LIN {X -0.046,Y -453.549,Z 733.557,A 0.000,B 0.000,C 90.000,E1 280.254} C_DIS
LIN {X 0.067,Y -465.639,Z 733.548,A 0.000,B 0.000,C 90.000,E1 278.690} C_DIS
LIN {X -0.179,Y -473.336,Z 733.543,A 0.000,B 0.000,C 90.000,E1 277.701} C_DIS
LIN {X -0.211,Y -478.457,Z 733.538,A 0.000,B 0.000,C 90.000,E1 276.947} C_DIS
LIN {X 0.222,Y -482.858,Z 733.534,A 0.000,B 0.000,C 90.000,E1 276.144} C_DIS
LIN {X -0.212,Y -486.445,Z 733.530,A 0.000,B 0.000,C 90.000,E1 275.448} C_DIS
LIN {X 0.102,Y -487.449,Z 733.529,A 0.000,B 0.000,C 90.000,E1 275.163} C_DIS
LIN {X -0.185,Y -489.129,Z 733.526,A 0.000,B 0.000,C 90.000,E1 274.702} C_DIS
LIN {X -0.017,Y -490.429,Z 733.523,A 0.000,B 0.000,C 90.000,E1 274.188} C_DIS
LIN {X 0.198,Y -491.326,Z 733.521,A 0.000,B 0.000,C 90.000,E1 273.669} C_DIS
LIN {X -0.101,Y -491.778,Z 733.518,A 0.000,B 0.000,C 90.000,E1 273.212} C_DIS
LIN {X 0.124,Y -491.880,Z 733.515,A 0.000,B 0.000,C 90.000,E1 272.694} C_DIS
LIN {X -0.164,Y -491.605,Z 733.512,A 0.000,B 0.000,C 90.000,E1 272.236} C_DIS
LIN {X 0.057,Y -490.893,Z 733.510,A 0.000,B 0.000,C 90.000,E1 271.718} C_DIS
LIN {X -0.231,Y -489.791,Z 733.507,A 0.000,B 0.000,C 90.000,E1 271.260} C_DIS
LIN {X -0.031,Y -488.272,Z 733.504,A 0.000,B 0.000,C 90.000,E1 270.745} C_DIS
LIN {X 0.162,Y -486.222,Z 733.501,A 0.000,B 0.000,C 90.000,E1 270.229} C_DIS
LIN {X -0.139,Y -483.595,Z 733.499,A 0.000,B 0.000,C 90.000,E1 269.771} C_DIS
LIN {X 0.026,Y -480.228,Z 733.496,A 0.000,B 0.000,C 90.000,E1 269.255} C_DIS
LIN {X 0.171,Y -476.025,Z 733.493,A 0.000,B 0.000,C 90.000,E1 268.740} C_DIS
LIN {X -0.006,Y -473.521,Z 733.492,A 0.000,B 0.000,C 90.000,E1 268.511} C_DIS
LIN {X -0.139,Y -467.895,Z 733.489,A 0.000,B 0.000,C 90.000,E1 268.051} C_DIS
LIN {X 0.151,Y -461.751,Z 733.487,A 0.000,B 0.000,C 90.000,E1 267.593} C_DIS
LIN {X 0.008,Y -455.030,Z 733.485,A 0.000,B 0.000,C 90.000,E1 267.249} C_DIS
LIN {X -0.087,Y -447.759,Z 733.483,A 0.000,B 0.000,C 90.000,E1 266.963} C_DIS
LIN {X -0.124,Y -439.978,Z 733.482,A 0.000,B 0.000,C 90.000,E1 266.731} C_DIS
LIN {X -0.126,Y -431.439,Z 733.481,A 0.000,B 0.000,C 90.000,E1 266.560} C_DIS
LIN {X 0.048,Y -423.516,Z 733.480,A 0.000,B 0.000,C 90.000,E1 266.445} C_DIS
LIN {X -0.116,Y -418.864,Z 733.480,A 0.000,B 0.000,C 90.000,E1 266.445} C_DIS
LIN {X -0.086,Y -180.942,Z 733.480,A 0.000,B 0.000,C 90.000,E1 266.445} C_DIS
LIN {X -0.075,Y -180.767,Z 733.471,A 0.000,B 0.000,C 90.000,E1 264.723} C_DIS
LIN {X -0.004,Y -178.861,Z 733.442,A 0.000,B 0.000,C 90.000,E1 259.634} C_DIS
LIN {X 0.067,Y -175.904,Z 733.414,A 0.000,B 0.000,C 90.000,E1 254.519} C_DIS
LIN {X 0.006,Y -174.587,Z 733.405,A 0.000,B 0.000,C 90.000,E1 252.834} C_DIS
LIN {X 0.041,Y -171.570,Z 733.381,A 0.000,B 0.000,C 90.000,E1 248.539} C_DIS
LIN {X 0.023,Y -167.793,Z 733.357,A 0.000,B 0.000,C 90.000,E1 244.229} C_DIS
LIN {X 0.037,Y -166.509,Z 733.347,A 0.000,B 0.000,C 90.000,E1 242.487} C_DIS
LIN {X 0.032,Y -163.218,Z 733.328,A 0.000,B 0.000,C 90.000,E1 238.997} C_DIS
LIN {X -0.003,Y -161.183,Z 733.313,A 0.000,B 0.000,C 90.000,E1 236.373} C_DIS
LIN {X -0.003,Y -157.196,Z 733.289,A 0.000,B 0.000,C 90.000,E1 231.949} C_DIS
LIN {X 0.043,Y -155.924,Z 733.279,A 0.000,B 0.000,C 90.000,E1 230.150} C_DIS
LIN {X -0.007,Y -152.175,Z 733.254,A 0.000,B 0.000,C 90.000,E1 225.688} C_DIS
LIN {X 0.008,Y -150.423,Z 733.239,A 0.000,B 0.000,C 90.000,E1 222.975} C_DIS
LIN {X -0.066,Y -147.151,Z 733.214,A 0.000,B 0.000,C 90.000,E1 218.463} C_DIS
LIN {X 0.021,Y -145.165,Z 733.193,A 0.000,B 0.000,C 90.000,E1 214.771} C_DIS
LIN {X -0.063,Y -142.318,Z 733.163,A 0.000,B 0.000,C 90.000,E1 209.283} C_DIS
LIN {X 0.058,Y -141.708,Z 733.152,A 0.000,B 0.000,C 90.000,E1 207.385} C_DIS
LIN {X -0.020,Y -139.470,Z 733.116,A 0.000,B 0.000,C 90.000,E1 200.918} C_DIS
LIN {X 0.034,Y -139.202,Z 733.106,A 0.000,B 0.000,C 90.000,E1 199.033} C_DIS
LIN {X -0.039,Y -138.329,Z 733.054,A 0.000,B 0.000,C 90.000,E1 189.726} C_DIS
LIN {X -0.036,Y -139.441,Z 733.007,A 0.000,B 0.000,C 90.000,E1 181.318} C_DIS
LIN {X 0.043,Y -140.976,Z 732.976,A 0.000,B 0.000,C 90.000,E1 175.698} C_DIS
LIN {X -0.007,Y -142.731,Z 732.956,A 0.000,B 0.000,C 90.000,E1 172.008} C_DIS
LIN {X -0.050,Y -145.119,Z 732.930,A 0.000,B 0.000,C 90.000,E1 167.409} C_DIS
LIN {X -0.055,Y -147.743,Z 732.910,A 0.000,B 0.000,C 90.000,E1 163.740} C_DIS
LIN {X 0.026,Y -150.409,Z 732.889,A 0.000,B 0.000,C 90.000,E1 160.061} C_DIS
LIN {X 0.042,Y -153.847,Z 732.869,A 0.000,B 0.000,C 90.000,E1 156.433} C_DIS
LIN {X -0.041,Y -157.258,Z 732.849,A 0.000,B 0.000,C 90.000,E1 152.871} C_DIS
LIN {X 0.037,Y -161.432,Z 732.829,A 0.000,B 0.000,C 90.000,E1 149.282} C_DIS
LIN {X 0.044,Y -165.633,Z 732.810,A 0.000,B 0.000,C 90.000,E1 145.754} C_DIS
LIN {X 0.027,Y -170.564,Z 732.790,A 0.000,B 0.000,C 90.000,E1 142.271} C_DIS
LIN {X -0.065,Y -175.443,Z 732.771,A 0.000,B 0.000,C 90.000,E1 138.852} C_DIS
LIN {X 0.051,Y -181.066,Z 732.752,A 0.000,B 0.000,C 90.000,E1 135.405} C_DIS
LIN {X -0.084,Y -186.504,Z 732.734,A 0.000,B 0.000,C 90.000,E1 132.081} C_DIS
LIN {X 0.015,Y -191.572,Z 732.718,A 0.000,B 0.000,C 90.000,E1 129.277} C_DIS
LIN {X -0.056,Y -191.740,Z 732.718,A 0.000,B 0.000,C 90.000,E1 129.197} C_DIS
LIN {X -0.129,Y -290.705,Z 732.718,A 0.000,B 0.000,C 90.000,E1 129.197} C_DIS
LIN {X 0.010,Y -291.831,Z 732.718,A 0.000,B 0.000,C 90.000,E1 129.152} C_DIS
LIN {X -0.060,Y -296.587,Z 732.716,A 0.000,B 0.000,C 90.000,E1 128.955} C_DIS
LIN {X -0.089,Y -299.097,Z 732.715,A 0.000,B 0.000,C 90.000,E1 128.749} C_DIS
LIN {X -0.093,Y -302.912,Z 732.712,A 0.000,B 0.000,C 90.000,E1 128.257} C_DIS
LIN {X 0.096,Y -304.694,Z 732.711,A 0.000,B 0.000,C 90.000,E1 127.890} C_DIS
LIN {X 0.042,Y -306.088,Z 732.709,A 0.000,B 0.000,C 90.000,E1 127.569} C_DIS
LIN {X -0.168,Y -309.945,Z 732.701,A 0.000,B 0.000,C 90.000,E1 126.297} C_DIS
LIN {X -0.051,Y -320.114,Z 732.683,A 0.000,B 0.000,C 90.000,E1 123.038} C_DIS
LIN {X -0.047,Y -330.586,Z 732.668,A 0.000,B 0.000,C 90.000,E1 120.178} C_DIS
LIN {X -0.131,Y -342.421,Z 732.652,A 0.000,B 0.000,C 90.000,E1 117.385} C_DIS
LIN {X -0.181,Y -355.717,Z 732.637,A 0.000,B 0.000,C 90.000,E1 114.643} C_DIS
LIN {X 0.103,Y -368.862,Z 732.623,A 0.000,B 0.000,C 90.000,E1 112.206} C_DIS
LIN {X -0.031,Y -383.352,Z 732.610,A 0.000,B 0.000,C 90.000,E1 109.885} C_DIS
LIN {X 0.074,Y -399.291,Z 732.598,A 0.000,B 0.000,C 90.000,E1 107.583} C_DIS
LIN {X -0.051,Y -416.796,Z 732.585,A 0.000,B 0.000,C 90.000,E1 105.371} C_DIS
LIN {X 0.159,Y -435.964,Z 732.573,A 0.000,B 0.000,C 90.000,E1 103.175} C_DIS
LIN {X -0.137,Y -456.118,Z 732.562,A 0.000,B 0.000,C 90.000,E1 101.186} C_DIS
LIN {X 0.211,Y -468.863,Z 732.555,A 0.000,B 0.000,C 90.000,E1 99.962} C_DIS
LIN {X 0.182,Y -470.793,Z 732.554,A 0.000,B 0.000,C 90.000,E1 99.726} C_DIS
LIN {X 0.073,Y -472.261,Z 732.553,A 0.000,B 0.000,C 90.000,E1 99.500} C_DIS
LIN {X 0.252,Y -474.285,Z 732.550,A 0.000,B 0.000,C 90.000,E1 98.973} C_DIS
LIN {X -0.104,Y -475.176,Z 732.547,A 0.000,B 0.000,C 90.000,E1 98.511} C_DIS
LIN {X 0.022,Y -475.088,Z 732.544,A 0.000,B 0.000,C 90.000,E1 97.992} C_DIS
LIN {X 0.156,Y -474.014,Z 732.542,A 0.000,B 0.000,C 90.000,E1 97.473} C_DIS
LIN {X 0.018,Y -473.060,Z 732.540,A 0.000,B 0.000,C 90.000,E1 97.239} C_DIS
LIN {X -0.122,Y -471.768,Z 732.539,A 0.000,B 0.000,C 90.000,E1 97.004} C_DIS
LIN {X 0.005,Y -453.891,Z 732.523,A 0.000,B 0.000,C 90.000,E1 94.188} C_DIS
LIN {X -0.165,Y -439.054,Z 732.509,A 0.000,B 0.000,C 90.000,E1 91.604} C_DIS
LIN {X -0.208,Y -431.544,Z 732.501,A 0.000,B 0.000,C 90.000,E1 90.286} C_DIS
LIN {X 0.015,Y -419.099,Z 732.490,A 0.000,B 0.000,C 90.000,E1 88.108} C_DIS
LIN {X -0.140,Y -408.057,Z 732.479,A 0.000,B 0.000,C 90.000,E1 86.216} C_DIS
LIN {X -0.063,Y -396.902,Z 732.468,A 0.000,B 0.000,C 90.000,E1 84.261} C_DIS
LIN {X -0.132,Y -384.313,Z 732.456,A 0.000,B 0.000,C 90.000,E1 82.008} C_DIS
LIN {X -0.068,Y -372.095,Z 732.443,A 0.000,B 0.000,C 90.000,E1 79.690} C_DIS
LIN {X -0.123,Y -358.888,Z 732.428,A 0.000,B 0.000,C 90.000,E1 77.048} C_DIS
LIN {X -0.046,Y -348.945,Z 732.416,A 0.000,B 0.000,C 90.000,E1 74.936} C_DIS
LIN {X -0.032,Y -336.383,Z 732.401,A 0.000,B 0.000,C 90.000,E1 72.181} C_DIS
LIN {X -0.140,Y -324.350,Z 732.385,A 0.000,B 0.000,C 90.000,E1 69.390} C_DIS
LIN {X -0.011,Y -312.017,Z 732.368,A 0.000,B 0.000,C 90.000,E1 66.177} C_DIS
LIN {X -0.012,Y -301.168,Z 732.350,A 0.000,B 0.000,C 90.000,E1 62.922} C_DIS
LIN {X -0.049,Y -291.225,Z 732.331,A 0.000,B 0.000,C 90.000,E1 59.616} C_DIS
LIN {X -0.008,Y -283.697,Z 732.316,A 0.000,B 0.000,C 90.000,E1 56.914} C_DIS
LIN {X -0.076,Y -276.550,Z 732.301,A 0.000,B 0.000,C 90.000,E1 54.196} C_DIS
LIN {X -0.001,Y -269.411,Z 732.286,A 0.000,B 0.000,C 90.000,E1 51.412} C_DIS
LIN {X 0.051,Y -263.888,Z 732.274,A 0.000,B 0.000,C 90.000,E1 49.299} C_DIS
LIN {X 0.067,Y -256.395,Z 732.258,A 0.000,B 0.000,C 90.000,E1 46.458} C_DIS
LIN {X -0.145,Y -250.679,Z 732.246,A 0.000,B 0.000,C 90.000,E1 44.352} C_DIS
LIN {X 0.068,Y -244.854,Z 732.234,A 0.000,B 0.000,C 90.000,E1 42.123} C_DIS
LIN {X 0.019,Y -238.963,Z 732.222,A 0.000,B 0.000,C 90.000,E1 39.930} C_DIS
LIN {X -0.061,Y -229.499,Z 732.201,A 0.000,B 0.000,C 90.000,E1 36.217} C_DIS
LIN {X -0.085,Y -220.772,Z 732.180,A 0.000,B 0.000,C 90.000,E1 32.418} C_DIS
LIN {X 0.074,Y -214.464,Z 732.163,A 0.000,B 0.000,C 90.000,E1 29.283} C_DIS
LIN {X 0.044,Y -208.878,Z 732.145,A 0.000,B 0.000,C 90.000,E1 26.155} C_DIS
LIN {X -0.032,Y -202.897,Z 732.123,A 0.000,B 0.000,C 90.000,E1 22.206} C_DIS
LIN {X -0.018,Y -198.172,Z 732.101,A 0.000,B 0.000,C 90.000,E1 18.181} C_DIS
LIN {X -0.014,Y -194.509,Z 732.078,A 0.000,B 0.000,C 90.000,E1 14.120} C_DIS
LIN {X -0.020,Y -191.545,Z 732.051,A 0.000,B 0.000,C 90.000,E1 9.208} C_DIS
LIN {X -0.029,Y -191.025,Z 731.974,A 0.000,B 0.000,C 90.000,E1 355.412} C_DIS
LIN {X 0.080,Y -193.620,Z 731.947,A 0.000,B 0.000,C 90.000,E1 350.443} C_DIS
LIN {X 0.087,Y -196.990,Z 731.924,A 0.000,B 0.000,C 90.000,E1 346.353} C_DIS
LIN {X 0.047,Y -201.312,Z 731.902,A 0.000,B 0.000,C 90.000,E1 342.308} C_DIS
LIN {X 0.073,Y -206.533,Z 731.879,A 0.000,B 0.000,C 90.000,E1 338.284} C_DIS
LIN {X 0.008,Y -212.775,Z 731.857,A 0.000,B 0.000,C 90.000,E1 334.332} C_DIS
LIN {X 0.027,Y -219.597,Z 731.836,A 0.000,B 0.000,C 90.000,E1 330.411} C_DIS
LIN {X 0.046,Y -227.020,Z 731.814,A 0.000,B 0.000,C 90.000,E1 326.548} C_DIS
LIN {X -0.007,Y -235.102,Z 731.793,A 0.000,B 0.000,C 90.000,E1 322.763} C_DIS
LIN {X 0.058,Y -243.917,Z 731.772,A 0.000,B 0.000,C 90.000,E1 319.013} C_DIS
LIN {X -0.021,Y -253.550,Z 731.752,A 0.000,B 0.000,C 90.000,E1 315.364} C_DIS
LIN {X 0.055,Y -264.373,Z 731.732,A 0.000,B 0.000,C 90.000,E1 311.757} C_DIS
LIN {X -0.002,Y -276.186,Z 731.713,A 0.000,B 0.000,C 90.000,E1 308.257} C_DIS
LIN {X 0.030,Y -289.374,Z 731.693,A 0.000,B 0.000,C 90.000,E1 304.818} C_DIS
LIN {X 0.067,Y -304.184,Z 731.675,A 0.000,B 0.000,C 90.000,E1 301.465} C_DIS
LIN {X -0.087,Y -315.631,Z 731.662,A 0.000,B 0.000,C 90.000,E1 299.205} C_DIS
LIN {X 0.145,Y -333.522,Z 731.644,A 0.000,B 0.000,C 90.000,E1 295.976} C_DIS
LIN {X 0.052,Y -350.964,Z 731.629,A 0.000,B 0.000,C 90.000,E1 293.206} C_DIS
LIN {X -0.120,Y -373.760,Z 731.611,A 0.000,B 0.000,C 90.000,E1 289.939} C_DIS
LIN {X 0.126,Y -392.212,Z 731.598,A 0.000,B 0.000,C 90.000,E1 287.583} C_DIS
LIN {X 0.054,Y -406.448,Z 731.588,A 0.000,B 0.000,C 90.000,E1 285.898} C_DIS
LIN {X 0.012,Y -420.554,Z 731.579,A 0.000,B 0.000,C 90.000,E1 284.245} C_DIS
LIN {X 0.082,Y -432.003,Z 731.572,A 0.000,B 0.000,C 90.000,E1 282.883} C_DIS
LIN {X 0.200,Y -442.999,Z 731.564,A 0.000,B 0.000,C 90.000,E1 281.535} C_DIS
LIN {X -0.051,Y -453.387,Z 731.557,A 0.000,B 0.000,C 90.000,E1 280.254} C_DIS
LIN {X 0.130,Y -465.479,Z 731.548,A 0.000,B 0.000,C 90.000,E1 278.681} C_DIS
LIN {X -0.190,Y -473.188,Z 731.543,A 0.000,B 0.000,C 90.000,E1 277.701} C_DIS
LIN {X 0.253,Y -478.317,Z 731.538,A 0.000,B 0.000,C 90.000,E1 276.891} C_DIS
LIN {X 0.209,Y -482.707,Z 731.534,A 0.000,B 0.000,C 90.000,E1 276.144} C_DIS
LIN {X 0.258,Y -486.253,Z 731.530,A 0.000,B 0.000,C 90.000,E1 275.391} C_DIS
LIN {X 0.087,Y -487.248,Z 731.529,A 0.000,B 0.000,C 90.000,E1 275.163} C_DIS
LIN {X -0.200,Y -488.920,Z 731.526,A 0.000,B 0.000,C 90.000,E1 274.702} C_DIS
LIN {X -0.035,Y -490.200,Z 731.523,A 0.000,B 0.000,C 90.000,E1 274.188} C_DIS
LIN {X 0.180,Y -491.070,Z 731.521,A 0.000,B 0.000,C 90.000,E1 273.669} C_DIS
LIN {X -0.120,Y -491.497,Z 731.518,A 0.000,B 0.000,C 90.000,E1 273.212} C_DIS
LIN {X 0.103,Y -491.580,Z 731.515,A 0.000,B 0.000,C 90.000,E1 272.694} C_DIS
LIN {X -0.187,Y -491.309,Z 731.512,A 0.000,B 0.000,C 90.000,E1 272.236} C_DIS
LIN {X 0.033,Y -490.597,Z 731.510,A 0.000,B 0.000,C 90.000,E1 271.718} C_DIS
LIN {X 0.233,Y -489.509,Z 731.507,A 0.000,B 0.000,C 90.000,E1 271.203} C_DIS
LIN {X -0.059,Y -488.013,Z 731.504,A 0.000,B 0.000,C 90.000,E1 270.745} C_DIS
LIN {X 0.133,Y -486.001,Z 731.501,A 0.000,B 0.000,C 90.000,E1 270.229} C_DIS
LIN {X -0.168,Y -483.404,Z 731.499,A 0.000,B 0.000,C 90.000,E1 269.771} C_DIS
LIN {X -0.004,Y -480.098,Z 731.496,A 0.000,B 0.000,C 90.000,E1 269.255} C_DIS
LIN {X 0.139,Y -475.872,Z 731.493,A 0.000,B 0.000,C 90.000,E1 268.740} C_DIS
LIN {X -0.213,Y -470.568,Z 731.490,A 0.000,B 0.000,C 90.000,E1 268.282} C_DIS
LIN {X -0.220,Y -467.738,Z 731.489,A 0.000,B 0.000,C 90.000,E1 268.051} C_DIS
LIN {X 0.044,Y -461.530,Z 731.487,A 0.000,B 0.000,C 90.000,E1 267.593} C_DIS
LIN {X -0.109,Y -454.863,Z 731.485,A 0.000,B 0.000,C 90.000,E1 267.249} C_DIS
LIN {X -0.084,Y -451.037,Z 731.484,A 0.000,B 0.000,C 90.000,E1 267.078} C_DIS
LIN {X 0.095,Y -443.345,Z 731.482,A 0.000,B 0.000,C 90.000,E1 266.788} C_DIS
LIN {X -0.147,Y -434.887,Z 731.481,A 0.000,B 0.000,C 90.000,E1 266.617} C_DIS
LIN {X 0.128,Y -425.733,Z 731.480,A 0.000,B 0.000,C 90.000,E1 266.445} C_DIS
LIN {X -0.198,Y -419.011,Z 731.480,A 0.000,B 0.000,C 90.000,E1 266.445} C_DIS
LIN {X 0.060,Y -180.942,Z 731.480,A 0.000,B 0.000,C 90.000,E1 266.388} C_DIS
LIN {X 0.071,Y -180.762,Z 731.470,A 0.000,B 0.000,C 90.000,E1 264.666} C_DIS
LIN {X -0.038,Y -178.856,Z 731.442,A 0.000,B 0.000,C 90.000,E1 259.634} C_DIS
LIN {X 0.034,Y -175.900,Z 731.414,A 0.000,B 0.000,C 90.000,E1 254.519} C_DIS
LIN {X -0.027,Y -174.578,Z 731.405,A 0.000,B 0.000,C 90.000,E1 252.834} C_DIS
LIN {X 0.007,Y -171.561,Z 731.381,A 0.000,B 0.000,C 90.000,E1 248.539} C_DIS
LIN {X -0.010,Y -167.785,Z 731.357,A 0.000,B 0.000,C 90.000,E1 244.229} C_DIS
LIN {X 0.005,Y -166.499,Z 731.347,A 0.000,B 0.000,C 90.000,E1 242.487} C_DIS
LIN {X 0.000,Y -163.208,Z 731.328,A 0.000,B 0.000,C 90.000,E1 238.997} C_DIS
LIN {X -0.035,Y -161.172,Z 731.313,A 0.000,B 0.000,C 90.000,E1 236.373} C_DIS
LIN {X 0.089,Y -157.186,Z 731.289,A 0.000,B 0.000,C 90.000,E1 231.904} C_DIS
LIN {X 0.012,Y -155.916,Z 731.279,A 0.000,B 0.000,C 90.000,E1 230.150} C_DIS
LIN {X 0.069,Y -152.167,Z 731.254,A 0.000,B 0.000,C 90.000,E1 225.648} C_DIS
LIN {X -0.023,Y -150.415,Z 731.239,A 0.000,B 0.000,C 90.000,E1 222.975} C_DIS
LIN {X 0.019,Y -147.144,Z 731.214,A 0.000,B 0.000,C 90.000,E1 218.418} C_DIS
LIN {X 0.016,Y -145.703,Z 731.198,A 0.000,B 0.000,C 90.000,E1 215.678} C_DIS
LIN {X 0.023,Y -143.085,Z 731.173,A 0.000,B 0.000,C 90.000,E1 211.082} C_DIS
LIN {X 0.029,Y -141.703,Z 731.152,A 0.000,B 0.000,C 90.000,E1 207.385} C_DIS
LIN {X -0.049,Y -139.468,Z 731.116,A 0.000,B 0.000,C 90.000,E1 200.918} C_DIS
LIN {X 0.005,Y -139.201,Z 731.106,A 0.000,B 0.000,C 90.000,E1 199.033} C_DIS
LIN {X 0.068,Y -138.328,Z 731.054,A 0.000,B 0.000,C 90.000,E1 189.670} C_DIS
LIN {X -0.066,Y -139.443,Z 731.007,A 0.000,B 0.000,C 90.000,E1 181.318} C_DIS
LIN {X 0.014,Y -140.981,Z 730.976,A 0.000,B 0.000,C 90.000,E1 175.698} C_DIS
LIN {X -0.036,Y -142.736,Z 730.956,A 0.000,B 0.000,C 90.000,E1 172.008} C_DIS
LIN {X 0.062,Y -145.127,Z 730.930,A 0.000,B 0.000,C 90.000,E1 167.353} C_DIS
LIN {X 0.056,Y -147.750,Z 730.909,A 0.000,B 0.000,C 90.000,E1 163.685} C_DIS
LIN {X -0.004,Y -150.419,Z 730.889,A 0.000,B 0.000,C 90.000,E1 160.061} C_DIS
LIN {X 0.010,Y -153.859,Z 730.869,A 0.000,B 0.000,C 90.000,E1 156.433} C_DIS
LIN {X -0.072,Y -157.270,Z 730.849,A 0.000,B 0.000,C 90.000,E1 152.871} C_DIS
LIN {X 0.005,Y -161.447,Z 730.829,A 0.000,B 0.000,C 90.000,E1 149.282} C_DIS
LIN {X 0.012,Y -165.648,Z 730.810,A 0.000,B 0.000,C 90.000,E1 145.754} C_DIS
LIN {X -0.006,Y -170.581,Z 730.790,A 0.000,B 0.000,C 90.000,E1 142.271} C_DIS
LIN {X -0.099,Y -175.459,Z 730.771,A 0.000,B 0.000,C 90.000,E1 138.852} C_DIS
LIN {X 0.016,Y -181.082,Z 730.752,A 0.000,B 0.000,C 90.000,E1 135.405} C_DIS
LIN {X 0.007,Y -186.523,Z 730.734,A 0.000,B 0.000,C 90.000,E1 132.043} C_DIS
LIN {X -0.020,Y -191.589,Z 730.718,A 0.000,B 0.000,C 90.000,E1 129.277} C_DIS
LIN {X 0.007,Y -191.708,Z 730.718,A 0.000,B 0.000,C 90.000,E1 129.197} C_DIS
LIN {X -0.024,Y -290.454,Z 730.718,A 0.000,B 0.000,C 90.000,E1 129.197} C_DIS
LIN {X 0.143,Y -292.896,Z 730.717,A 0.000,B 0.000,C 90.000,E1 129.116} C_DIS
LIN {X 0.116,Y -296.939,Z 730.716,A 0.000,B 0.000,C 90.000,E1 128.910} C_DIS
LIN {X -0.144,Y -299.327,Z 730.715,A 0.000,B 0.000,C 90.000,E1 128.749} C_DIS
LIN {X -0.075,Y -303.151,Z 730.712,A 0.000,B 0.000,C 90.000,E1 128.222} C_DIS
LIN {X -0.073,Y -304.863,Z 730.710,A 0.000,B 0.000,C 90.000,E1 127.890} C_DIS
LIN {X 0.116,Y -306.203,Z 730.709,A 0.000,B 0.000,C 90.000,E1 127.523} C_DIS
LIN {X -0.018,Y -314.920,Z 730.692,A 0.000,B 0.000,C 90.000,E1 124.612} C_DIS
LIN {X 0.102,Y -325.861,Z 730.674,A 0.000,B 0.000,C 90.000,E1 121.386} C_DIS
LIN {X 0.052,Y -337.094,Z 730.659,A 0.000,B 0.000,C 90.000,E1 118.565} C_DIS
LIN {X 0.018,Y -349.741,Z 730.643,A 0.000,B 0.000,C 90.000,E1 115.796} C_DIS
LIN {X -0.027,Y -362.264,Z 730.630,A 0.000,B 0.000,C 90.000,E1 113.387} C_DIS
LIN {X -0.196,Y -376.086,Z 730.617,A 0.000,B 0.000,C 90.000,E1 111.046} C_DIS
LIN {X -0.155,Y -391.304,Z 730.604,A 0.000,B 0.000,C 90.000,E1 108.725} C_DIS
LIN {X 0.019,Y -408.030,Z 730.591,A 0.000,B 0.000,C 90.000,E1 106.441} C_DIS
LIN {X -0.006,Y -426.384,Z 730.579,A 0.000,B 0.000,C 90.000,E1 104.245} C_DIS
LIN {X 0.128,Y -446.191,Z 730.567,A 0.000,B 0.000,C 90.000,E1 102.119} C_DIS
LIN {X 0.022,Y -469.054,Z 730.555,A 0.000,B 0.000,C 90.000,E1 99.962} C_DIS
LIN {X -0.025,Y -470.957,Z 730.554,A 0.000,B 0.000,C 90.000,E1 99.726} C_DIS
LIN {X -0.152,Y -472.403,Z 730.553,A 0.000,B 0.000,C 90.000,E1 99.500} C_DIS
LIN {X 0.027,Y -474.369,Z 730.550,A 0.000,B 0.000,C 90.000,E1 98.973} C_DIS
LIN {X 0.141,Y -475.214,Z 730.547,A 0.000,B 0.000,C 90.000,E1 98.454} C_DIS
LIN {X -0.203,Y -475.082,Z 730.544,A 0.000,B 0.000,C 90.000,E1 97.992} C_DIS
LIN {X -0.006,Y -473.962,Z 730.541,A 0.000,B 0.000,C 90.000,E1 97.466} C_DIS
LIN {X -0.206,Y -472.980,Z 730.540,A 0.000,B 0.000,C 90.000,E1 97.239} C_DIS
LIN {X 0.122,Y -471.654,Z 730.539,A 0.000,B 0.000,C 90.000,E1 96.947} C_DIS
LIN {X 0.040,Y -452.227,Z 730.522,A 0.000,B 0.000,C 90.000,E1 93.898} C_DIS
LIN {X 0.059,Y -438.929,Z 730.509,A 0.000,B 0.000,C 90.000,E1 91.547} C_DIS
LIN {X 0.010,Y -431.419,Z 730.501,A 0.000,B 0.000,C 90.000,E1 90.229} C_DIS
LIN {X 0.095,Y -420.536,Z 730.491,A 0.000,B 0.000,C 90.000,E1 88.339} C_DIS
LIN {X -0.097,Y -411.123,Z 730.482,A 0.000,B 0.000,C 90.000,E1 86.731} C_DIS
LIN {X 0.015,Y -400.009,Z 730.471,A 0.000,B 0.000,C 90.000,E1 84.780} C_DIS
LIN {X -0.038,Y -388.917,Z 730.460,A 0.000,B 0.000,C 90.000,E1 82.818} C_DIS
LIN {X 0.089,Y -375.106,Z 730.446,A 0.000,B 0.000,C 90.000,E1 80.218} C_DIS
LIN {X -0.004,Y -360.315,Z 730.429,A 0.000,B 0.000,C 90.000,E1 77.297} C_DIS
LIN {X 0.199,Y -348.938,Z 730.416,A 0.000,B 0.000,C 90.000,E1 74.866} C_DIS
LIN {X 0.112,Y -336.392,Z 730.401,A 0.000,B 0.000,C 90.000,E1 72.127} C_DIS
LIN {X -0.006,Y -324.388,Z 730.385,A 0.000,B 0.000,C 90.000,E1 69.337} C_DIS
LIN {X -0.098,Y -313.255,Z 730.369,A 0.000,B 0.000,C 90.000,E1 66.485} C_DIS
LIN {X -0.090,Y -303.370,Z 730.353,A 0.000,B 0.000,C 90.000,E1 63.563} C_DIS
LIN {X -0.050,Y -293.340,Z 730.335,A 0.000,B 0.000,C 90.000,E1 60.255} C_DIS
LIN {X -0.099,Y -285.776,Z 730.320,A 0.000,B 0.000,C 90.000,E1 57.582} C_DIS
LIN {X 0.022,Y -276.791,Z 730.301,A 0.000,B 0.000,C 90.000,E1 54.149} C_DIS
LIN {X 0.082,Y -271.470,Z 730.289,A 0.000,B 0.000,C 90.000,E1 52.065} C_DIS
LIN {X 0.000,Y -266.029,Z 730.278,A 0.000,B 0.000,C 90.000,E1 49.989} C_DIS
LIN {X -0.011,Y -260.411,Z 730.266,A 0.000,B 0.000,C 90.000,E1 47.877} C_DIS
LIN {X 0.030,Y -254.806,Z 730.254,A 0.000,B 0.000,C 90.000,E1 45.729} C_DIS
LIN {X -0.028,Y -249.029,Z 730.242,A 0.000,B 0.000,C 90.000,E1 43.581} C_DIS
LIN {X -0.012,Y -243.173,Z 730.230,A 0.000,B 0.000,C 90.000,E1 41.391} C_DIS
LIN {X -0.124,Y -235.311,Z 730.214,A 0.000,B 0.000,C 90.000,E1 38.463} C_DIS
LIN {X -0.076,Y -226.129,Z 730.193,A 0.000,B 0.000,C 90.000,E1 34.692} C_DIS
LIN {X 0.077,Y -219.325,Z 730.176,A 0.000,B 0.000,C 90.000,E1 31.592} C_DIS
LIN {X 0.083,Y -213.153,Z 730.158,A 0.000,B 0.000,C 90.000,E1 28.487} C_DIS
LIN {X 0.109,Y -207.762,Z 730.141,A 0.000,B 0.000,C 90.000,E1 25.335} C_DIS
LIN {X -0.071,Y -203.043,Z 730.123,A 0.000,B 0.000,C 90.000,E1 22.206} C_DIS
LIN {X -0.053,Y -198.302,Z 730.101,A 0.000,B 0.000,C 90.000,E1 18.181} C_DIS
LIN {X -0.044,Y -194.624,Z 730.078,A 0.000,B 0.000,C 90.000,E1 14.120} C_DIS
LIN {X -0.046,Y -191.640,Z 730.051,A 0.000,B 0.000,C 90.000,E1 9.208} C_DIS
LIN {X 0.044,Y -190.829,Z 729.979,A 0.000,B 0.000,C 90.000,E1 356.216} C_DIS
LIN {X 0.088,Y -193.734,Z 729.947,A 0.000,B 0.000,C 90.000,E1 350.443} C_DIS
LIN {X -0.094,Y -197.092,Z 729.924,A 0.000,B 0.000,C 90.000,E1 346.408} C_DIS
LIN {X 0.061,Y -201.422,Z 729.902,A 0.000,B 0.000,C 90.000,E1 342.308} C_DIS
LIN {X 0.092,Y -206.646,Z 729.880,A 0.000,B 0.000,C 90.000,E1 338.284} C_DIS
LIN {X 0.030,Y -212.868,Z 729.857,A 0.000,B 0.000,C 90.000,E1 334.332} C_DIS
LIN {X 0.053,Y -219.668,Z 729.836,A 0.000,B 0.000,C 90.000,E1 330.411} C_DIS
LIN {X -0.050,Y -227.083,Z 729.814,A 0.000,B 0.000,C 90.000,E1 326.580} C_DIS
LIN {X 0.026,Y -235.146,Z 729.793,A 0.000,B 0.000,C 90.000,E1 322.763} C_DIS
LIN {X 0.093,Y -243.941,Z 729.772,A 0.000,B 0.000,C 90.000,E1 319.013} C_DIS
LIN {X 0.016,Y -253.569,Z 729.752,A 0.000,B 0.000,C 90.000,E1 315.364} C_DIS
LIN {X 0.101,Y -264.377,Z 729.732,A 0.000,B 0.000,C 90.000,E1 311.757} C_DIS
LIN {X 0.046,Y -276.193,Z 729.713,A 0.000,B 0.000,C 90.000,E1 308.257} C_DIS
LIN {X 0.081,Y -289.396,Z 729.694,A 0.000,B 0.000,C 90.000,E1 304.818} C_DIS
LIN {X 0.121,Y -304.202,Z 729.675,A 0.000,B 0.000,C 90.000,E1 301.465} C_DIS
LIN {X 0.025,Y -317.366,Z 729.660,A 0.000,B 0.000,C 90.000,E1 298.871} C_DIS
LIN {X -0.132,Y -335.357,Z 729.643,A 0.000,B 0.000,C 90.000,E1 295.720} C_DIS
LIN {X 0.143,Y -352.888,Z 729.627,A 0.000,B 0.000,C 90.000,E1 292.898} C_DIS
LIN {X -0.057,Y -373.658,Z 729.611,A 0.000,B 0.000,C 90.000,E1 289.939} C_DIS
LIN {X -0.036,Y -394.432,Z 729.596,A 0.000,B 0.000,C 90.000,E1 287.330} C_DIS
LIN {X -0.193,Y -408.645,Z 729.587,A 0.000,B 0.000,C 90.000,E1 285.662} C_DIS
LIN {X 0.074,Y -420.364,Z 729.579,A 0.000,B 0.000,C 90.000,E1 284.245} C_DIS
LIN {X -0.132,Y -434.067,Z 729.570,A 0.000,B 0.000,C 90.000,E1 282.647} C_DIS
LIN {X 0.003,Y -444.904,Z 729.563,A 0.000,B 0.000,C 90.000,E1 281.299} C_DIS
LIN {X 0.227,Y -455.218,Z 729.555,A 0.000,B 0.000,C 90.000,E1 279.962} C_DIS
LIN {X -0.087,Y -467.277,Z 729.547,A 0.000,B 0.000,C 90.000,E1 278.454} C_DIS
LIN {X -0.172,Y -473.012,Z 729.543,A 0.000,B 0.000,C 90.000,E1 277.701} C_DIS
LIN {X -0.205,Y -478.134,Z 729.538,A 0.000,B 0.000,C 90.000,E1 276.947} C_DIS
LIN {X 0.224,Y -482.540,Z 729.534,A 0.000,B 0.000,C 90.000,E1 276.144} C_DIS
LIN {X -0.085,Y -484.988,Z 729.531,A 0.000,B 0.000,C 90.000,E1 275.682} C_DIS
LIN {X 0.101,Y -487.038,Z 729.529,A 0.000,B 0.000,C 90.000,E1 275.163} C_DIS
LIN {X -0.189,Y -488.729,Z 729.526,A 0.000,B 0.000,C 90.000,E1 274.702} C_DIS
LIN {X -0.023,Y -489.945,Z 729.523,A 0.000,B 0.000,C 90.000,E1 274.188} C_DIS
LIN {X 0.190,Y -490.796,Z 729.521,A 0.000,B 0.000,C 90.000,E1 273.669} C_DIS
LIN {X -0.111,Y -491.226,Z 729.518,A 0.000,B 0.000,C 90.000,E1 273.212} C_DIS
LIN {X 0.110,Y -491.287,Z 729.515,A 0.000,B 0.000,C 90.000,E1 272.694} C_DIS
LIN {X -0.181,Y -491.001,Z 729.512,A 0.000,B 0.000,C 90.000,E1 272.236} C_DIS
LIN {X 0.036,Y -490.313,Z 729.510,A 0.000,B 0.000,C 90.000,E1 271.718} C_DIS
LIN {X 0.235,Y -489.271,Z 729.507,A 0.000,B 0.000,C 90.000,E1 271.203} C_DIS
LIN {X -0.058,Y -487.780,Z 729.504,A 0.000,B 0.000,C 90.000,E1 270.745} C_DIS
LIN {X 0.133,Y -485.791,Z 729.501,A 0.000,B 0.000,C 90.000,E1 270.229} C_DIS
LIN {X -0.170,Y -483.220,Z 729.499,A 0.000,B 0.000,C 90.000,E1 269.771} C_DIS
LIN {X -0.008,Y -479.950,Z 729.496,A 0.000,B 0.000,C 90.000,E1 269.255} C_DIS
LIN {X 0.135,Y -475.738,Z 729.493,A 0.000,B 0.000,C 90.000,E1 268.740} C_DIS
LIN {X -0.218,Y -470.492,Z 729.490,A 0.000,B 0.000,C 90.000,E1 268.282} C_DIS
LIN {X -0.226,Y -467.713,Z 729.489,A 0.000,B 0.000,C 90.000,E1 268.051} C_DIS
LIN {X 0.003,Y -461.493,Z 729.487,A 0.000,B 0.000,C 90.000,E1 267.593} C_DIS
LIN {X -0.174,Y -454.747,Z 729.485,A 0.000,B 0.000,C 90.000,E1 267.249} C_DIS
LIN {X -0.140,Y -450.972,Z 729.484,A 0.000,B 0.000,C 90.000,E1 267.078} C_DIS
LIN {X 0.027,Y -443.244,Z 729.482,A 0.000,B 0.000,C 90.000,E1 266.788} C_DIS
LIN {X -0.194,Y -434.968,Z 729.481,A 0.000,B 0.000,C 90.000,E1 266.617} C_DIS
LIN {X 0.065,Y -425.951,Z 729.480,A 0.000,B 0.000,C 90.000,E1 266.445} C_DIS
LIN {X 0.149,Y -419.361,Z 729.480,A 0.000,B 0.000,C 90.000,E1 266.388} C_DIS
LIN {X 0.029,Y -180.942,Z 729.480,A 0.000,B 0.000,C 90.000,E1 266.388} C_DIS
LIN {X 0.037,Y -180.758,Z 729.470,A 0.000,B 0.000,C 90.000,E1 264.666} C_DIS
LIN {X -0.072,Y -178.851,Z 729.442,A 0.000,B 0.000,C 90.000,E1 259.634} C_DIS
LIN {X 0.000,Y -175.895,Z 729.414,A 0.000,B 0.000,C 90.000,E1 254.519} C_DIS
LIN {X -0.061,Y -174.568,Z 729.405,A 0.000,B 0.000,C 90.000,E1 252.834} C_DIS
LIN {X -0.025,Y -171.553,Z 729.381,A 0.000,B 0.000,C 90.000,E1 248.539} C_DIS
LIN {X 0.030,Y -167.777,Z 729.357,A 0.000,B 0.000,C 90.000,E1 244.204} C_DIS
LIN {X -0.028,Y -166.488,Z 729.347,A 0.000,B 0.000,C 90.000,E1 242.487} C_DIS
LIN {X -0.031,Y -163.199,Z 729.328,A 0.000,B 0.000,C 90.000,E1 238.997} C_DIS
LIN {X 0.023,Y -161.162,Z 729.313,A 0.000,B 0.000,C 90.000,E1 236.342} C_DIS
LIN {X 0.057,Y -157.178,Z 729.288,A 0.000,B 0.000,C 90.000,E1 231.904} C_DIS
LIN {X -0.019,Y -155.908,Z 729.279,A 0.000,B 0.000,C 90.000,E1 230.150} C_DIS
LIN {X 0.038,Y -152.158,Z 729.254,A 0.000,B 0.000,C 90.000,E1 225.648} C_DIS
LIN {X 0.058,Y -150.408,Z 729.239,A 0.000,B 0.000,C 90.000,E1 222.933} C_DIS
LIN {X 0.081,Y -147.137,Z 729.213,A 0.000,B 0.000,C 90.000,E1 218.382} C_DIS
LIN {X -0.014,Y -145.698,Z 729.198,A 0.000,B 0.000,C 90.000,E1 215.678} C_DIS
LIN {X -0.007,Y -143.080,Z 729.173,A 0.000,B 0.000,C 90.000,E1 211.082} C_DIS
LIN {X -0.001,Y -141.699,Z 729.152,A 0.000,B 0.000,C 90.000,E1 207.385} C_DIS
LIN {X -0.078,Y -139.465,Z 729.116,A 0.000,B 0.000,C 90.000,E1 200.918} C_DIS
LIN {X -0.024,Y -139.198,Z 729.106,A 0.000,B 0.000,C 90.000,E1 199.033} C_DIS
LIN {X 0.040,Y -138.327,Z 729.054,A 0.000,B 0.000,C 90.000,E1 189.670} C_DIS
LIN {X 0.044,Y -139.447,Z 729.007,A 0.000,B 0.000,C 90.000,E1 181.260} C_DIS
LIN {X -0.015,Y -140.985,Z 728.976,A 0.000,B 0.000,C 90.000,E1 175.698} C_DIS
LIN {X -0.066,Y -142.741,Z 728.955,A 0.000,B 0.000,C 90.000,E1 172.008} C_DIS
LIN {X 0.033,Y -145.134,Z 728.930,A 0.000,B 0.000,C 90.000,E1 167.353} C_DIS
LIN {X 0.026,Y -147.758,Z 728.909,A 0.000,B 0.000,C 90.000,E1 163.685} C_DIS
LIN {X -0.035,Y -150.428,Z 728.889,A 0.000,B 0.000,C 90.000,E1 160.061} C_DIS
LIN {X -0.021,Y -153.871,Z 728.869,A 0.000,B 0.000,C 90.000,E1 156.433} C_DIS
LIN {X 0.036,Y -157.282,Z 728.849,A 0.000,B 0.000,C 90.000,E1 152.820} C_DIS
LIN {X -0.027,Y -161.461,Z 728.829,A 0.000,B 0.000,C 90.000,E1 149.282} C_DIS
LIN {X -0.021,Y -165.662,Z 728.810,A 0.000,B 0.000,C 90.000,E1 145.754} C_DIS
LIN {X -0.039,Y -170.599,Z 728.790,A 0.000,B 0.000,C 90.000,E1 142.271} C_DIS
LIN {X -0.001,Y -175.476,Z 728.771,A 0.000,B 0.000,C 90.000,E1 138.809} C_DIS
LIN {X -0.019,Y -181.098,Z 728.752,A 0.000,B 0.000,C 90.000,E1 135.405} C_DIS
LIN {X -0.029,Y -186.541,Z 728.734,A 0.000,B 0.000,C 90.000,E1 132.043} C_DIS
LIN {X -0.054,Y -191.606,Z 728.718,A 0.000,B 0.000,C 90.000,E1 129.277} C_DIS
LIN {X 0.059,Y -191.682,Z 728.718,A 0.000,B 0.000,C 90.000,E1 129.197} C_DIS
LIN {X 0.042,Y -290.697,Z 728.718,A 0.000,B 0.000,C 90.000,E1 129.197} C_DIS
LIN {X -0.009,Y -296.805,Z 728.716,A 0.000,B 0.000,C 90.000,E1 128.955} C_DIS
LIN {X 0.034,Y -299.506,Z 728.715,A 0.000,B 0.000,C 90.000,E1 128.705} C_DIS
LIN {X 0.077,Y -303.270,Z 728.712,A 0.000,B 0.000,C 90.000,E1 128.177} C_DIS
LIN {X 0.026,Y -304.941,Z 728.710,A 0.000,B 0.000,C 90.000,E1 127.855} C_DIS
LIN {X 0.030,Y -306.253,Z 728.708,A 0.000,B 0.000,C 90.000,E1 127.523} C_DIS
LIN {X 0.188,Y -317.017,Z 728.689,A 0.000,B 0.000,C 90.000,E1 123.913} C_DIS
LIN {X 0.107,Y -327.081,Z 728.673,A 0.000,B 0.000,C 90.000,E1 121.052} C_DIS
LIN {X 0.096,Y -338.471,Z 728.657,A 0.000,B 0.000,C 90.000,E1 118.231} C_DIS
LIN {X 0.093,Y -351.294,Z 728.642,A 0.000,B 0.000,C 90.000,E1 115.463} C_DIS
LIN {X -0.063,Y -363.981,Z 728.628,A 0.000,B 0.000,C 90.000,E1 113.078} C_DIS
LIN {X -0.190,Y -377.980,Z 728.615,A 0.000,B 0.000,C 90.000,E1 110.737} C_DIS
LIN {X -0.103,Y -393.391,Z 728.602,A 0.000,B 0.000,C 90.000,E1 108.417} C_DIS
LIN {X 0.120,Y -410.323,Z 728.590,A 0.000,B 0.000,C 90.000,E1 106.134} C_DIS
LIN {X 0.043,Y -428.902,Z 728.578,A 0.000,B 0.000,C 90.000,E1 103.953} C_DIS
LIN {X -0.107,Y -448.835,Z 728.566,A 0.000,B 0.000,C 90.000,E1 101.883} C_DIS
LIN {X -0.077,Y -469.144,Z 728.555,A 0.000,B 0.000,C 90.000,E1 99.962} C_DIS
LIN {X -0.133,Y -471.038,Z 728.554,A 0.000,B 0.000,C 90.000,E1 99.726} C_DIS
LIN {X 0.198,Y -472.474,Z 728.553,A 0.000,B 0.000,C 90.000,E1 99.443} C_DIS
LIN {X -0.089,Y -474.418,Z 728.550,A 0.000,B 0.000,C 90.000,E1 98.973} C_DIS
LIN {X 0.024,Y -475.244,Z 728.547,A 0.000,B 0.000,C 90.000,E1 98.454} C_DIS
LIN {X 0.152,Y -475.096,Z 728.544,A 0.000,B 0.000,C 90.000,E1 97.936} C_DIS
LIN {X -0.122,Y -473.956,Z 728.541,A 0.000,B 0.000,C 90.000,E1 97.466} C_DIS
LIN {X 0.148,Y -472.962,Z 728.540,A 0.000,B 0.000,C 90.000,E1 97.182} C_DIS
LIN {X 0.008,Y -471.623,Z 728.539,A 0.000,B 0.000,C 90.000,E1 96.947} C_DIS
LIN {X -0.072,Y -452.179,Z 728.522,A 0.000,B 0.000,C 90.000,E1 93.898} C_DIS
LIN {X -0.050,Y -438.882,Z 728.509,A 0.000,B 0.000,C 90.000,E1 91.547} C_DIS
LIN {X -0.097,Y -431.368,Z 728.501,A 0.000,B 0.000,C 90.000,E1 90.229} C_DIS
LIN {X -0.011,Y -420.515,Z 728.491,A 0.000,B 0.000,C 90.000,E1 88.339} C_DIS
LIN {X 0.209,Y -411.111,Z 728.482,A 0.000,B 0.000,C 90.000,E1 86.674} C_DIS
LIN {X -0.009,Y -398.423,Z 728.469,A 0.000,B 0.000,C 90.000,E1 84.489} C_DIS
LIN {X -0.091,Y -385.792,Z 728.457,A 0.000,B 0.000,C 90.000,E1 82.243} C_DIS
LIN {X 0.003,Y -373.616,Z 728.444,A 0.000,B 0.000,C 90.000,E1 79.926} C_DIS
LIN {X -0.050,Y -358.922,Z 728.428,A 0.000,B 0.000,C 90.000,E1 76.992} C_DIS
LIN {X 0.042,Y -347.596,Z 728.414,A 0.000,B 0.000,C 90.000,E1 74.574} C_DIS
LIN {X 0.031,Y -336.480,Z 728.401,A 0.000,B 0.000,C 90.000,E1 72.127} C_DIS
LIN {X -0.080,Y -324.497,Z 728.385,A 0.000,B 0.000,C 90.000,E1 69.337} C_DIS
LIN {X -0.169,Y -313.388,Z 728.369,A 0.000,B 0.000,C 90.000,E1 66.485} C_DIS
LIN {X 0.119,Y -303.548,Z 728.353,A 0.000,B 0.000,C 90.000,E1 63.512} C_DIS
LIN {X -0.105,Y -293.565,Z 728.335,A 0.000,B 0.000,C 90.000,E1 60.255} C_DIS
LIN {X 0.093,Y -286.024,Z 728.320,A 0.000,B 0.000,C 90.000,E1 57.533} C_DIS
LIN {X -0.016,Y -277.085,Z 728.301,A 0.000,B 0.000,C 90.000,E1 54.149} C_DIS
LIN {X 0.021,Y -270.005,Z 728.285,A 0.000,B 0.000,C 90.000,E1 51.376} C_DIS
LIN {X -0.082,Y -264.503,Z 728.274,A 0.000,B 0.000,C 90.000,E1 49.299} C_DIS
LIN {X -0.047,Y -257.028,Z 728.258,A 0.000,B 0.000,C 90.000,E1 46.458} C_DIS
LIN {X 0.110,Y -251.315,Z 728.246,A 0.000,B 0.000,C 90.000,E1 44.271} C_DIS
LIN {X -0.018,Y -245.464,Z 728.234,A 0.000,B 0.000,C 90.000,E1 42.123} C_DIS
LIN {X -0.054,Y -239.528,Z 728.222,A 0.000,B 0.000,C 90.000,E1 39.930} C_DIS
LIN {X -0.041,Y -231.832,Z 728.205,A 0.000,B 0.000,C 90.000,E1 36.950} C_DIS
LIN {X -0.050,Y -222.892,Z 728.184,A 0.000,B 0.000,C 90.000,E1 33.166} C_DIS
LIN {X -0.025,Y -216.347,Z 728.167,A 0.000,B 0.000,C 90.000,E1 30.079} C_DIS
LIN {X 0.000,Y -210.528,Z 728.150,A 0.000,B 0.000,C 90.000,E1 26.950} C_DIS
LIN {X -0.036,Y -204.323,Z 728.128,A 0.000,B 0.000,C 90.000,E1 23.003} C_DIS
LIN {X -0.077,Y -200.223,Z 728.110,A 0.000,B 0.000,C 90.000,E1 19.812} C_DIS
LIN {X 0.047,Y -196.116,Z 728.087,A 0.000,B 0.000,C 90.000,E1 15.733} C_DIS
LIN {X 0.037,Y -192.574,Z 728.060,A 0.000,B 0.000,C 90.000,E1 10.838} C_DIS
LIN {X 0.077,Y -190.203,Z 728.024,A 0.000,B 0.000,C 90.000,E1 4.245} C_DIS
LIN {X -0.089,Y -191.573,Z 727.970,A 0.000,B 0.000,C 90.000,E1 354.609} C_DIS
LIN {X 0.062,Y -194.450,Z 727.943,A 0.000,B 0.000,C 90.000,E1 349.634} C_DIS
LIN {X -0.013,Y -197.993,Z 727.920,A 0.000,B 0.000,C 90.000,E1 345.574} C_DIS
LIN {X 0.043,Y -202.517,Z 727.897,A 0.000,B 0.000,C 90.000,E1 341.511} C_DIS
LIN {X -0.080,Y -207.921,Z 727.875,A 0.000,B 0.000,C 90.000,E1 337.539} C_DIS
LIN {X -0.015,Y -214.268,Z 727.853,A 0.000,B 0.000,C 90.000,E1 333.563} C_DIS
LIN {X -0.036,Y -221.187,Z 727.831,A 0.000,B 0.000,C 90.000,E1 329.665} C_DIS
LIN {X 0.036,Y -228.704,Z 727.810,A 0.000,B 0.000,C 90.000,E1 325.801} C_DIS
LIN {X -0.016,Y -236.871,Z 727.789,A 0.000,B 0.000,C 90.000,E1 322.029} C_DIS
LIN {X -0.082,Y -245.807,Z 727.768,A 0.000,B 0.000,C 90.000,E1 318.324} C_DIS
LIN {X -0.104,Y -255.638,Z 727.748,A 0.000,B 0.000,C 90.000,E1 314.676} C_DIS
LIN {X -0.004,Y -265.508,Z 727.730,A 0.000,B 0.000,C 90.000,E1 311.434} C_DIS
LIN {X -0.033,Y -277.469,Z 727.711,A 0.000,B 0.000,C 90.000,E1 307.935} C_DIS
LIN {X 0.100,Y -290.838,Z 727.692,A 0.000,B 0.000,C 90.000,E1 304.485} C_DIS
LIN {X -0.068,Y -305.808,Z 727.673,A 0.000,B 0.000,C 90.000,E1 301.180} C_DIS
LIN {X -0.011,Y -319.091,Z 727.659,A 0.000,B 0.000,C 90.000,E1 298.565} C_DIS
LIN {X -0.106,Y -337.210,Z 727.641,A 0.000,B 0.000,C 90.000,E1 295.412} C_DIS
LIN {X -0.129,Y -352.837,Z 727.627,A 0.000,B 0.000,C 90.000,E1 292.950} C_DIS
LIN {X 0.091,Y -375.772,Z 727.609,A 0.000,B 0.000,C 90.000,E1 289.631} C_DIS
LIN {X 0.019,Y -394.289,Z 727.596,A 0.000,B 0.000,C 90.000,E1 287.330} C_DIS
LIN {X -0.139,Y -408.473,Z 727.587,A 0.000,B 0.000,C 90.000,E1 285.662} C_DIS
LIN {X 0.126,Y -420.137,Z 727.579,A 0.000,B 0.000,C 90.000,E1 284.245} C_DIS
LIN {X 0.160,Y -431.586,Z 727.572,A 0.000,B 0.000,C 90.000,E1 282.883} C_DIS
LIN {X -0.160,Y -442.597,Z 727.564,A 0.000,B 0.000,C 90.000,E1 281.591} C_DIS
LIN {X 0.019,Y -452.984,Z 727.557,A 0.000,B 0.000,C 90.000,E1 280.254} C_DIS
LIN {X 0.123,Y -465.066,Z 727.548,A 0.000,B 0.000,C 90.000,E1 278.690} C_DIS
LIN {X -0.129,Y -472.785,Z 727.543,A 0.000,B 0.000,C 90.000,E1 277.701} C_DIS
LIN {X -0.163,Y -477.935,Z 727.539,A 0.000,B 0.000,C 90.000,E1 276.947} C_DIS
LIN {X -0.215,Y -482.343,Z 727.534,A 0.000,B 0.000,C 90.000,E1 276.201} C_DIS
LIN {X -0.047,Y -484.789,Z 727.532,A 0.000,B 0.000,C 90.000,E1 275.682} C_DIS
LIN {X 0.138,Y -486.854,Z 727.529,A 0.000,B 0.000,C 90.000,E1 275.163} C_DIS
LIN {X -0.150,Y -488.496,Z 727.526,A 0.000,B 0.000,C 90.000,E1 274.702} C_DIS
LIN {X 0.014,Y -489.733,Z 727.523,A 0.000,B 0.000,C 90.000,E1 274.188} C_DIS
LIN {X 0.225,Y -490.531,Z 727.521,A 0.000,B 0.000,C 90.000,E1 273.669} C_DIS
LIN {X -0.077,Y -490.975,Z 727.518,A 0.000,B 0.000,C 90.000,E1 273.212} C_DIS
LIN {X 0.143,Y -491.016,Z 727.515,A 0.000,B 0.000,C 90.000,E1 272.694} C_DIS
LIN {X -0.150,Y -490.695,Z 727.512,A 0.000,B 0.000,C 90.000,E1 272.236} C_DIS
LIN {X 0.066,Y -490.046,Z 727.510,A 0.000,B 0.000,C 90.000,E1 271.718} C_DIS
LIN {X -0.226,Y -489.013,Z 727.507,A 0.000,B 0.000,C 90.000,E1 271.260} C_DIS
LIN {X -0.032,Y -487.543,Z 727.504,A 0.000,B 0.000,C 90.000,E1 270.745} C_DIS
LIN {X 0.157,Y -485.581,Z 727.501,A 0.000,B 0.000,C 90.000,E1 270.229} C_DIS
LIN {X -0.147,Y -483.025,Z 727.499,A 0.000,B 0.000,C 90.000,E1 269.771} C_DIS
LIN {X 0.015,Y -479.786,Z 727.496,A 0.000,B 0.000,C 90.000,E1 269.255} C_DIS
LIN {X -0.154,Y -477.852,Z 727.495,A 0.000,B 0.000,C 90.000,E1 269.026} C_DIS
LIN {X -0.021,Y -473.221,Z 727.492,A 0.000,B 0.000,C 90.000,E1 268.511} C_DIS
LIN {X -0.219,Y -467.650,Z 727.489,A 0.000,B 0.000,C 90.000,E1 268.051} C_DIS
LIN {X 0.210,Y -464.516,Z 727.488,A 0.000,B 0.000,C 90.000,E1 267.764} C_DIS
LIN {X 0.149,Y -457.899,Z 727.485,A 0.000,B 0.000,C 90.000,E1 267.364} C_DIS
LIN {X 0.195,Y -450.645,Z 727.484,A 0.000,B 0.000,C 90.000,E1 267.020} C_DIS
LIN {X -0.053,Y -443.125,Z 727.482,A 0.000,B 0.000,C 90.000,E1 266.788} C_DIS
LIN {X 0.136,Y -434.690,Z 727.481,A 0.000,B 0.000,C 90.000,E1 266.560} C_DIS
LIN {X -0.044,Y -425.457,Z 727.480,A 0.000,B 0.000,C 90.000,E1 266.445} C_DIS
LIN {X 0.046,Y -417.581,Z 727.480,A 0.000,B 0.000,C 90.000,E1 266.388} C_DIS
LIN {X -0.016,Y -180.940,Z 727.480,A 0.000,B 0.000,C 90.000,E1 266.388} C_DIS
LIN {X -0.007,Y -180.752,Z 727.470,A 0.000,B 0.000,C 90.000,E1 264.666} C_DIS
LIN {X 0.061,Y -178.845,Z 727.442,A 0.000,B 0.000,C 90.000,E1 259.577} C_DIS
LIN {X -0.042,Y -175.889,Z 727.414,A 0.000,B 0.000,C 90.000,E1 254.519} C_DIS
LIN {X 0.064,Y -174.557,Z 727.404,A 0.000,B 0.000,C 90.000,E1 252.779} C_DIS
LIN {X -0.067,Y -171.541,Z 727.381,A 0.000,B 0.000,C 90.000,E1 248.539} C_DIS
LIN {X -0.011,Y -167.766,Z 727.357,A 0.000,B 0.000,C 90.000,E1 244.204} C_DIS
LIN {X -0.069,Y -166.474,Z 727.347,A 0.000,B 0.000,C 90.000,E1 242.487} C_DIS
LIN {X -0.072,Y -163.187,Z 727.328,A 0.000,B 0.000,C 90.000,E1 238.997} C_DIS
LIN {X -0.017,Y -161.149,Z 727.313,A 0.000,B 0.000,C 90.000,E1 236.342} C_DIS
LIN {X 0.018,Y -157.167,Z 727.288,A 0.000,B 0.000,C 90.000,E1 231.904} C_DIS
LIN {X 0.041,Y -155.898,Z 727.279,A 0.000,B 0.000,C 90.000,E1 230.114} C_DIS
LIN {X -0.001,Y -152.149,Z 727.254,A 0.000,B 0.000,C 90.000,E1 225.648} C_DIS
LIN {X 0.019,Y -150.398,Z 727.239,A 0.000,B 0.000,C 90.000,E1 222.933} C_DIS
LIN {X 0.042,Y -147.128,Z 727.213,A 0.000,B 0.000,C 90.000,E1 218.382} C_DIS
LIN {X 0.033,Y -145.690,Z 727.198,A 0.000,B 0.000,C 90.000,E1 215.644} C_DIS
LIN {X 0.030,Y -143.073,Z 727.173,A 0.000,B 0.000,C 90.000,E1 211.052} C_DIS
LIN {X -0.038,Y -141.693,Z 727.152,A 0.000,B 0.000,C 90.000,E1 207.385} C_DIS
LIN {X 0.016,Y -139.463,Z 727.116,A 0.000,B 0.000,C 90.000,E1 200.865} C_DIS
LIN {X -0.061,Y -139.196,Z 727.106,A 0.000,B 0.000,C 90.000,E1 199.033} C_DIS
LIN {X 0.002,Y -138.326,Z 727.054,A 0.000,B 0.000,C 90.000,E1 189.670} C_DIS
LIN {X 0.008,Y -139.449,Z 727.007,A 0.000,B 0.000,C 90.000,E1 181.260} C_DIS
LIN {X -0.053,Y -140.992,Z 726.976,A 0.000,B 0.000,C 90.000,E1 175.698} C_DIS
LIN {X 0.038,Y -142.747,Z 726.955,A 0.000,B 0.000,C 90.000,E1 171.951} C_DIS
LIN {X -0.005,Y -145.144,Z 726.930,A 0.000,B 0.000,C 90.000,E1 167.353} C_DIS
LIN {X -0.013,Y -147.767,Z 726.909,A 0.000,B 0.000,C 90.000,E1 163.685} C_DIS
LIN {X -0.074,Y -150.441,Z 726.889,A 0.000,B 0.000,C 90.000,E1 160.061} C_DIS
LIN {X 0.002,Y -153.887,Z 726.869,A 0.000,B 0.000,C 90.000,E1 156.410} C_DIS
LIN {X -0.004,Y -157.297,Z 726.849,A 0.000,B 0.000,C 90.000,E1 152.820} C_DIS
LIN {X 0.015,Y -161.481,Z 726.829,A 0.000,B 0.000,C 90.000,E1 149.253} C_DIS
LIN {X 0.031,Y -165.680,Z 726.810,A 0.000,B 0.000,C 90.000,E1 145.722} C_DIS
LIN {X -0.081,Y -170.620,Z 726.790,A 0.000,B 0.000,C 90.000,E1 142.271} C_DIS
LIN {X 0.072,Y -175.498,Z 726.771,A 0.000,B 0.000,C 90.000,E1 138.771} C_DIS
LIN {X -0.062,Y -181.118,Z 726.752,A 0.000,B 0.000,C 90.000,E1 135.405} C_DIS
LIN {X 0.066,Y -186.566,Z 726.733,A 0.000,B 0.000,C 90.000,E1 132.000} C_DIS
LIN {X -0.022,Y -191.519,Z 726.718,A 0.000,B 0.000,C 90.000,E1 129.322} C_DIS
LIN {X 0.125,Y -191.650,Z 726.718,A 0.000,B 0.000,C 90.000,E1 129.197} C_DIS
LIN {X 0.154,Y -290.394,Z 726.718,A 0.000,B 0.000,C 90.000,E1 129.197} C_DIS
LIN {X -0.071,Y -292.661,Z 726.718,A 0.000,B 0.000,C 90.000,E1 129.197} C_DIS
LIN {X -0.077,Y -297.167,Z 726.716,A 0.000,B 0.000,C 90.000,E1 128.955} C_DIS
LIN {X -0.036,Y -299.735,Z 726.715,A 0.000,B 0.000,C 90.000,E1 128.705} C_DIS
LIN {X -0.110,Y -303.502,Z 726.712,A 0.000,B 0.000,C 90.000,E1 128.177} C_DIS
LIN {X 0.080,Y -305.105,Z 726.710,A 0.000,B 0.000,C 90.000,E1 127.810} C_DIS
LIN {X -0.158,Y -306.366,Z 726.708,A 0.000,B 0.000,C 90.000,E1 127.523} C_DIS
LIN {X 0.062,Y -318.166,Z 726.687,A 0.000,B 0.000,C 90.000,E1 123.579} C_DIS
LIN {X 0.015,Y -328.387,Z 726.671,A 0.000,B 0.000,C 90.000,E1 120.718} C_DIS
LIN {X 0.034,Y -339.949,Z 726.655,A 0.000,B 0.000,C 90.000,E1 117.897} C_DIS
LIN {X -0.081,Y -352.951,Z 726.640,A 0.000,B 0.000,C 90.000,E1 115.155} C_DIS
LIN {X -0.198,Y -365.815,Z 726.626,A 0.000,B 0.000,C 90.000,E1 112.770} C_DIS
LIN {X 0.073,Y -380.003,Z 726.613,A 0.000,B 0.000,C 90.000,E1 110.375} C_DIS
LIN {X 0.223,Y -395.615,Z 726.600,A 0.000,B 0.000,C 90.000,E1 108.055} C_DIS
LIN {X 0.006,Y -412.767,Z 726.588,A 0.000,B 0.000,C 90.000,E1 105.843} C_DIS
LIN {X 0.094,Y -431.584,Z 726.576,A 0.000,B 0.000,C 90.000,E1 103.647} C_DIS
LIN {X 0.028,Y -451.607,Z 726.564,A 0.000,B 0.000,C 90.000,E1 101.591} C_DIS
LIN {X 0.142,Y -466.995,Z 726.556,A 0.000,B 0.000,C 90.000,E1 100.141} C_DIS
LIN {X 0.176,Y -469.352,Z 726.555,A 0.000,B 0.000,C 90.000,E1 99.905} C_DIS
LIN {X 0.098,Y -471.220,Z 726.554,A 0.000,B 0.000,C 90.000,E1 99.670} C_DIS
LIN {X -0.060,Y -472.633,Z 726.552,A 0.000,B 0.000,C 90.000,E1 99.443} C_DIS
LIN {X 0.121,Y -474.512,Z 726.550,A 0.000,B 0.000,C 90.000,E1 98.916} C_DIS
LIN {X -0.233,Y -475.285,Z 726.547,A 0.000,B 0.000,C 90.000,E1 98.454} C_DIS
LIN {X -0.104,Y -475.087,Z 726.544,A 0.000,B 0.000,C 90.000,E1 97.936} C_DIS
LIN {X 0.092,Y -473.892,Z 726.541,A 0.000,B 0.000,C 90.000,E1 97.409} C_DIS
LIN {X -0.107,Y -472.865,Z 726.540,A 0.000,B 0.000,C 90.000,E1 97.182} C_DIS
LIN {X 0.222,Y -471.485,Z 726.538,A 0.000,B 0.000,C 90.000,E1 96.891} C_DIS
LIN {X -0.121,Y -453.562,Z 726.523,A 0.000,B 0.000,C 90.000,E1 94.131} C_DIS
LIN {X -0.031,Y -440.205,Z 726.510,A 0.000,B 0.000,C 90.000,E1 91.776} C_DIS
LIN {X -0.066,Y -432.732,Z 726.503,A 0.000,B 0.000,C 90.000,E1 90.458} C_DIS
LIN {X 0.054,Y -421.944,Z 726.492,A 0.000,B 0.000,C 90.000,E1 88.568} C_DIS
LIN {X -0.134,Y -412.569,Z 726.483,A 0.000,B 0.000,C 90.000,E1 86.963} C_DIS
LIN {X 0.080,Y -399.904,Z 726.471,A 0.000,B 0.000,C 90.000,E1 84.723} C_DIS
LIN {X 0.021,Y -388.834,Z 726.460,A 0.000,B 0.000,C 90.000,E1 82.761} C_DIS
LIN {X 0.214,Y -373.548,Z 726.444,A 0.000,B 0.000,C 90.000,E1 79.859} C_DIS
LIN {X 0.085,Y -358.880,Z 726.427,A 0.000,B 0.000,C 90.000,E1 76.937} C_DIS
LIN {X -0.168,Y -347.576,Z 726.414,A 0.000,B 0.000,C 90.000,E1 74.574} C_DIS
LIN {X -0.171,Y -336.487,Z 726.401,A 0.000,B 0.000,C 90.000,E1 72.127} C_DIS
LIN {X 0.099,Y -323.234,Z 726.383,A 0.000,B 0.000,C 90.000,E1 68.954} C_DIS
LIN {X -0.015,Y -312.297,Z 726.367,A 0.000,B 0.000,C 90.000,E1 66.102} C_DIS
LIN {X 0.188,Y -299.629,Z 726.346,A 0.000,B 0.000,C 90.000,E1 62.153} C_DIS
LIN {X -0.014,Y -289.929,Z 726.327,A 0.000,B 0.000,C 90.000,E1 58.869} C_DIS
LIN {X 0.084,Y -280.812,Z 726.308,A 0.000,B 0.000,C 90.000,E1 55.468} C_DIS
LIN {X 0.058,Y -275.571,Z 726.297,A 0.000,B 0.000,C 90.000,E1 53.417} C_DIS
LIN {X 0.097,Y -270.271,Z 726.285,A 0.000,B 0.000,C 90.000,E1 51.331} C_DIS
LIN {X -0.009,Y -264.772,Z 726.274,A 0.000,B 0.000,C 90.000,E1 49.256} C_DIS
LIN {X 0.014,Y -257.304,Z 726.258,A 0.000,B 0.000,C 90.000,E1 46.419} C_DIS
LIN {X 0.002,Y -251.581,Z 726.246,A 0.000,B 0.000,C 90.000,E1 44.271} C_DIS
LIN {X 0.064,Y -245.722,Z 726.234,A 0.000,B 0.000,C 90.000,E1 42.081} C_DIS
LIN {X 0.013,Y -237.800,Z 726.218,A 0.000,B 0.000,C 90.000,E1 39.152} C_DIS
LIN {X -0.012,Y -230.190,Z 726.201,A 0.000,B 0.000,C 90.000,E1 36.171} C_DIS
LIN {X 0.109,Y -221.358,Z 726.180,A 0.000,B 0.000,C 90.000,E1 32.339} C_DIS
LIN {X -0.020,Y -214.971,Z 726.163,A 0.000,B 0.000,C 90.000,E1 29.283} C_DIS
LIN {X -0.034,Y -209.355,Z 726.145,A 0.000,B 0.000,C 90.000,E1 26.155} C_DIS
LIN {X 0.093,Y -204.455,Z 726.128,A 0.000,B 0.000,C 90.000,E1 22.950} C_DIS
LIN {X 0.057,Y -200.360,Z 726.110,A 0.000,B 0.000,C 90.000,E1 19.758} C_DIS
LIN {X 0.051,Y -196.227,Z 726.087,A 0.000,B 0.000,C 90.000,E1 15.717} C_DIS
LIN {X -0.006,Y -192.683,Z 726.060,A 0.000,B 0.000,C 90.000,E1 10.838} C_DIS
LIN {X 0.038,Y -190.305,Z 726.024,A 0.000,B 0.000,C 90.000,E1 4.245} C_DIS
LIN {X -0.086,Y -191.695,Z 725.970,A 0.000,B 0.000,C 90.000,E1 354.609} C_DIS
LIN {X 0.070,Y -194.571,Z 725.943,A 0.000,B 0.000,C 90.000,E1 349.634} C_DIS
LIN {X -0.001,Y -198.102,Z 725.920,A 0.000,B 0.000,C 90.000,E1 345.574} C_DIS
LIN {X 0.059,Y -202.629,Z 725.897,A 0.000,B 0.000,C 90.000,E1 341.511} C_DIS
LIN {X -0.060,Y -208.030,Z 725.875,A 0.000,B 0.000,C 90.000,E1 337.539} C_DIS
LIN {X 0.010,Y -214.348,Z 725.853,A 0.000,B 0.000,C 90.000,E1 333.563} C_DIS
LIN {X -0.008,Y -221.244,Z 725.831,A 0.000,B 0.000,C 90.000,E1 329.665} C_DIS
LIN {X 0.009,Y -227.207,Z 725.814,A 0.000,B 0.000,C 90.000,E1 326.580} C_DIS
LIN {X 0.091,Y -235.213,Z 725.793,A 0.000,B 0.000,C 90.000,E1 322.763} C_DIS
LIN {X -0.022,Y -243.955,Z 725.773,A 0.000,B 0.000,C 90.000,E1 319.057} C_DIS
LIN {X -0.092,Y -253.595,Z 725.752,A 0.000,B 0.000,C 90.000,E1 315.405} C_DIS
LIN {X 0.177,Y -264.395,Z 725.732,A 0.000,B 0.000,C 90.000,E1 311.757} C_DIS
LIN {X -0.091,Y -276.235,Z 725.713,A 0.000,B 0.000,C 90.000,E1 308.302} C_DIS
LIN {X 0.167,Y -289.473,Z 725.694,A 0.000,B 0.000,C 90.000,E1 304.818} C_DIS
LIN {X -0.046,Y -304.268,Z 725.675,A 0.000,B 0.000,C 90.000,E1 301.514} C_DIS
LIN {X 0.038,Y -319.091,Z 725.659,A 0.000,B 0.000,C 90.000,E1 298.565} C_DIS
LIN {X -0.054,Y -337.193,Z 725.641,A 0.000,B 0.000,C 90.000,E1 295.412} C_DIS
LIN {X -0.076,Y -352.796,Z 725.627,A 0.000,B 0.000,C 90.000,E1 292.950} C_DIS
LIN {X 0.146,Y -375.667,Z 725.609,A 0.000,B 0.000,C 90.000,E1 289.631} C_DIS
LIN {X 0.120,Y -396.507,Z 725.595,A 0.000,B 0.000,C 90.000,E1 287.040} C_DIS
LIN {X 0.011,Y -410.649,Z 725.585,A 0.000,B 0.000,C 90.000,E1 285.371} C_DIS
LIN {X -0.097,Y -422.226,Z 725.578,A 0.000,B 0.000,C 90.000,E1 284.008} C_DIS
LIN {X -0.031,Y -433.627,Z 725.570,A 0.000,B 0.000,C 90.000,E1 282.647} C_DIS
LIN {X -0.111,Y -442.369,Z 725.564,A 0.000,B 0.000,C 90.000,E1 281.591} C_DIS
LIN {X 0.065,Y -452.760,Z 725.557,A 0.000,B 0.000,C 90.000,E1 280.254} C_DIS
LIN {X 0.002,Y -466.851,Z 725.547,A 0.000,B 0.000,C 90.000,E1 278.454} C_DIS
LIN {X 0.233,Y -474.400,Z 725.541,A 0.000,B 0.000,C 90.000,E1 277.409} C_DIS
LIN {X 0.152,Y -479.306,Z 725.537,A 0.000,B 0.000,C 90.000,E1 276.663} C_DIS
LIN {X 0.174,Y -483.448,Z 725.533,A 0.000,B 0.000,C 90.000,E1 275.910} C_DIS
LIN {X 0.176,Y -486.655,Z 725.529,A 0.000,B 0.000,C 90.000,E1 275.163} C_DIS
LIN {X -0.114,Y -488.281,Z 725.526,A 0.000,B 0.000,C 90.000,E1 274.702} C_DIS
LIN {X 0.050,Y -489.487,Z 725.523,A 0.000,B 0.000,C 90.000,E1 274.188} C_DIS
LIN {X -0.229,Y -490.291,Z 725.521,A 0.000,B 0.000,C 90.000,E1 273.726} C_DIS
LIN {X -0.044,Y -490.675,Z 725.518,A 0.000,B 0.000,C 90.000,E1 273.212} C_DIS
LIN {X 0.175,Y -490.721,Z 725.515,A 0.000,B 0.000,C 90.000,E1 272.694} C_DIS
LIN {X -0.119,Y -490.419,Z 725.512,A 0.000,B 0.000,C 90.000,E1 272.236} C_DIS
LIN {X 0.095,Y -489.763,Z 725.510,A 0.000,B 0.000,C 90.000,E1 271.718} C_DIS
LIN {X -0.199,Y -488.740,Z 725.507,A 0.000,B 0.000,C 90.000,E1 271.260} C_DIS
LIN {X -0.005,Y -487.299,Z 725.504,A 0.000,B 0.000,C 90.000,E1 270.745} C_DIS
LIN {X 0.181,Y -485.352,Z 725.501,A 0.000,B 0.000,C 90.000,E1 270.229} C_DIS
LIN {X -0.125,Y -482.831,Z 725.499,A 0.000,B 0.000,C 90.000,E1 269.771} C_DIS
LIN {X 0.035,Y -479.659,Z 725.496,A 0.000,B 0.000,C 90.000,E1 269.255} C_DIS
LIN {X 0.176,Y -475.582,Z 725.493,A 0.000,B 0.000,C 90.000,E1 268.740} C_DIS
LIN {X -0.178,Y -470.441,Z 725.490,A 0.000,B 0.000,C 90.000,E1 268.282} C_DIS
LIN {X 0.208,Y -464.464,Z 725.488,A 0.000,B 0.000,C 90.000,E1 267.764} C_DIS
LIN {X -0.050,Y -461.424,Z 725.487,A 0.000,B 0.000,C 90.000,E1 267.593} C_DIS
LIN {X 0.188,Y -454.622,Z 725.485,A 0.000,B 0.000,C 90.000,E1 267.192} C_DIS
LIN {X 0.069,Y -447.357,Z 725.483,A 0.000,B 0.000,C 90.000,E1 266.906} C_DIS
LIN {X 0.024,Y -439.612,Z 725.482,A 0.000,B 0.000,C 90.000,E1 266.674} C_DIS
LIN {X 0.000,Y -431.062,Z 725.481,A 0.000,B 0.000,C 90.000,E1 266.502} C_DIS
LIN {X 0.156,Y -423.177,Z 725.480,A 0.000,B 0.000,C 90.000,E1 266.388} C_DIS
LIN {X -0.011,Y -418.796,Z 725.480,A 0.000,B 0.000,C 90.000,E1 266.388} C_DIS
LIN {X -0.040,Y -180.940,Z 725.480,A 0.000,B 0.000,C 90.000,E1 266.388} C_DIS
LIN {X -0.031,Y -180.749,Z 725.470,A 0.000,B 0.000,C 90.000,E1 264.666} C_DIS
LIN {X 0.036,Y -178.841,Z 725.442,A 0.000,B 0.000,C 90.000,E1 259.577} C_DIS
LIN {X -0.067,Y -175.884,Z 725.414,A 0.000,B 0.000,C 90.000,E1 254.519} C_DIS
LIN {X 0.039,Y -174.550,Z 725.404,A 0.000,B 0.000,C 90.000,E1 252.779} C_DIS
LIN {X -0.028,Y -171.534,Z 725.381,A 0.000,B 0.000,C 90.000,E1 248.518} C_DIS
LIN {X -0.035,Y -167.760,Z 725.357,A 0.000,B 0.000,C 90.000,E1 244.204} C_DIS
LIN {X -0.092,Y -166.466,Z 725.347,A 0.000,B 0.000,C 90.000,E1 242.487} C_DIS
LIN {X 0.045,Y -163.180,Z 725.328,A 0.000,B 0.000,C 90.000,E1 238.948} C_DIS
LIN {X -0.041,Y -161.140,Z 725.313,A 0.000,B 0.000,C 90.000,E1 236.342} C_DIS
LIN {X -0.005,Y -157.161,Z 725.288,A 0.000,B 0.000,C 90.000,E1 231.904} C_DIS
LIN {X 0.019,Y -155.892,Z 725.278,A 0.000,B 0.000,C 90.000,E1 230.114} C_DIS
LIN {X -0.024,Y -152.143,Z 725.254,A 0.000,B 0.000,C 90.000,E1 225.648} C_DIS
LIN {X -0.003,Y -150.392,Z 725.239,A 0.000,B 0.000,C 90.000,E1 222.933} C_DIS
LIN {X 0.020,Y -147.123,Z 725.213,A 0.000,B 0.000,C 90.000,E1 218.382} C_DIS
LIN {X 0.011,Y -145.687,Z 725.198,A 0.000,B 0.000,C 90.000,E1 215.644} C_DIS
LIN {X 0.008,Y -143.069,Z 725.173,A 0.000,B 0.000,C 90.000,E1 211.052} C_DIS
LIN {X -0.059,Y -141.690,Z 725.152,A 0.000,B 0.000,C 90.000,E1 207.385} C_DIS
LIN {X -0.005,Y -139.461,Z 725.116,A 0.000,B 0.000,C 90.000,E1 200.865} C_DIS
LIN {X -0.037,Y -139.195,Z 725.106,A 0.000,B 0.000,C 90.000,E1 199.014} C_DIS
LIN {X -0.019,Y -138.325,Z 725.054,A 0.000,B 0.000,C 90.000,E1 189.670} C_DIS
LIN {X -0.014,Y -139.451,Z 725.007,A 0.000,B 0.000,C 90.000,E1 181.260} C_DIS
LIN {X 0.067,Y -140.996,Z 724.976,A 0.000,B 0.000,C 90.000,E1 175.641} C_DIS
LIN {X 0.016,Y -142.750,Z 724.955,A 0.000,B 0.000,C 90.000,E1 171.951} C_DIS
LIN {X -0.027,Y -145.150,Z 724.930,A 0.000,B 0.000,C 90.000,E1 167.353} C_DIS
LIN {X -0.034,Y -147.772,Z 724.909,A 0.000,B 0.000,C 90.000,E1 163.685} C_DIS
LIN {X 0.046,Y -150.448,Z 724.889,A 0.000,B 0.000,C 90.000,E1 160.007} C_DIS
LIN {X -0.020,Y -153.896,Z 724.869,A 0.000,B 0.000,C 90.000,E1 156.410} C_DIS
LIN {X -0.027,Y -157.306,Z 724.849,A 0.000,B 0.000,C 90.000,E1 152.820} C_DIS
LIN {X -0.008,Y -161.491,Z 724.829,A 0.000,B 0.000,C 90.000,E1 149.253} C_DIS
LIN {X 0.008,Y -165.691,Z 724.810,A 0.000,B 0.000,C 90.000,E1 145.722} C_DIS
LIN {X -0.105,Y -170.633,Z 724.790,A 0.000,B 0.000,C 90.000,E1 142.271} C_DIS
LIN {X 0.048,Y -175.509,Z 724.771,A 0.000,B 0.000,C 90.000,E1 138.771} C_DIS
LIN {X -0.087,Y -181.130,Z 724.752,A 0.000,B 0.000,C 90.000,E1 135.405} C_DIS
LIN {X 0.041,Y -186.579,Z 724.733,A 0.000,B 0.000,C 90.000,E1 132.000} C_DIS
LIN {X 0.006,Y -191.577,Z 724.718,A 0.000,B 0.000,C 90.000,E1 129.277} C_DIS
LIN {X -0.058,Y -191.608,Z 724.718,A 0.000,B 0.000,C 90.000,E1 129.277} C_DIS
LIN {X -0.137,Y -289.766,Z 724.718,A 0.000,B 0.000,C 90.000,E1 129.277} C_DIS
LIN {X -0.187,Y -290.886,Z 724.718,A 0.000,B 0.000,C 90.000,E1 129.277} C_DIS
LIN {X 0.053,Y -297.029,Z 724.716,A 0.000,B 0.000,C 90.000,E1 128.955} C_DIS
LIN {X 0.111,Y -299.906,Z 724.715,A 0.000,B 0.000,C 90.000,E1 128.669} C_DIS
LIN {X -0.182,Y -303.608,Z 724.712,A 0.000,B 0.000,C 90.000,E1 128.177} C_DIS
LIN {X 0.008,Y -305.171,Z 724.710,A 0.000,B 0.000,C 90.000,E1 127.810} C_DIS
LIN {X 0.200,Y -306.402,Z 724.708,A 0.000,B 0.000,C 90.000,E1 127.443} C_DIS
LIN {X -0.011,Y -318.189,Z 724.687,A 0.000,B 0.000,C 90.000,E1 123.579} C_DIS
LIN {X -0.059,Y -328.415,Z 724.671,A 0.000,B 0.000,C 90.000,E1 120.718} C_DIS
LIN {X -0.042,Y -339.984,Z 724.655,A 0.000,B 0.000,C 90.000,E1 117.897} C_DIS
LIN {X -0.159,Y -352.992,Z 724.640,A 0.000,B 0.000,C 90.000,E1 115.155} C_DIS
LIN {X 0.059,Y -365.862,Z 724.626,A 0.000,B 0.000,C 90.000,E1 112.717} C_DIS
LIN {X -0.009,Y -380.056,Z 724.613,A 0.000,B 0.000,C 90.000,E1 110.375} C_DIS
LIN {X 0.139,Y -395.677,Z 724.600,A 0.000,B 0.000,C 90.000,E1 108.055} C_DIS
LIN {X -0.080,Y -412.838,Z 724.588,A 0.000,B 0.000,C 90.000,E1 105.843} C_DIS
LIN {X 0.006,Y -431.664,Z 724.576,A 0.000,B 0.000,C 90.000,E1 103.647} C_DIS
LIN {X -0.058,Y -451.690,Z 724.564,A 0.000,B 0.000,C 90.000,E1 101.591} C_DIS
LIN {X 0.059,Y -467.081,Z 724.556,A 0.000,B 0.000,C 90.000,E1 100.141} C_DIS
LIN {X 0.093,Y -469.424,Z 724.555,A 0.000,B 0.000,C 90.000,E1 99.905} C_DIS
LIN {X 0.007,Y -471.285,Z 724.554,A 0.000,B 0.000,C 90.000,E1 99.670} C_DIS
LIN {X -0.081,Y -472.693,Z 724.552,A 0.000,B 0.000,C 90.000,E1 99.434} C_DIS
LIN {X 0.024,Y -474.554,Z 724.550,A 0.000,B 0.000,C 90.000,E1 98.916} C_DIS
LIN {X 0.140,Y -475.313,Z 724.547,A 0.000,B 0.000,C 90.000,E1 98.398} C_DIS
LIN {X -0.201,Y -475.102,Z 724.544,A 0.000,B 0.000,C 90.000,E1 97.936} C_DIS
LIN {X -0.005,Y -473.892,Z 724.541,A 0.000,B 0.000,C 90.000,E1 97.409} C_DIS
LIN {X -0.204,Y -472.855,Z 724.540,A 0.000,B 0.000,C 90.000,E1 97.182} C_DIS
LIN {X 0.126,Y -471.465,Z 724.538,A 0.000,B 0.000,C 90.000,E1 96.891} C_DIS
LIN {X -0.214,Y -453.535,Z 724.523,A 0.000,B 0.000,C 90.000,E1 94.131} C_DIS
LIN {X -0.122,Y -440.181,Z 724.510,A 0.000,B 0.000,C 90.000,E1 91.776} C_DIS
LIN {X -0.155,Y -432.725,Z 724.502,A 0.000,B 0.000,C 90.000,E1 90.458} C_DIS
LIN {X -0.034,Y -421.937,Z 724.492,A 0.000,B 0.000,C 90.000,E1 88.568} C_DIS
LIN {X 0.191,Y -412.563,Z 724.483,A 0.000,B 0.000,C 90.000,E1 86.906} C_DIS
LIN {X -0.053,Y -401.487,Z 724.472,A 0.000,B 0.000,C 90.000,E1 85.008} C_DIS
LIN {X -0.112,Y -390.435,Z 724.461,A 0.000,B 0.000,C 90.000,E1 83.053} C_DIS
LIN {X 0.129,Y -375.114,Z 724.445,A 0.000,B 0.000,C 90.000,E1 80.151} C_DIS
LIN {X 0.013,Y -358.961,Z 724.427,A 0.000,B 0.000,C 90.000,E1 76.937} C_DIS
LIN {X 0.120,Y -346.270,Z 724.412,A 0.000,B 0.000,C 90.000,E1 74.212} C_DIS
LIN {X 0.078,Y -335.236,Z 724.399,A 0.000,B 0.000,C 90.000,E1 71.764} C_DIS
LIN {X -0.050,Y -320.826,Z 724.380,A 0.000,B 0.000,C 90.000,E1 68.337} C_DIS
LIN {X -0.147,Y -311.330,Z 724.365,A 0.000,B 0.000,C 90.000,E1 65.793} C_DIS
LIN {X 0.144,Y -299.842,Z 724.345,A 0.000,B 0.000,C 90.000,E1 62.153} C_DIS
LIN {X -0.049,Y -290.184,Z 724.327,A 0.000,B 0.000,C 90.000,E1 58.869} C_DIS
LIN {X 0.058,Y -281.095,Z 724.308,A 0.000,B 0.000,C 90.000,E1 55.468} C_DIS
LIN {X 0.037,Y -275.871,Z 724.297,A 0.000,B 0.000,C 90.000,E1 53.417} C_DIS
LIN {X 0.082,Y -270.587,Z 724.285,A 0.000,B 0.000,C 90.000,E1 51.331} C_DIS
LIN {X -0.017,Y -265.128,Z 724.274,A 0.000,B 0.000,C 90.000,E1 49.256} C_DIS
LIN {X -0.066,Y -259.520,Z 724.262,A 0.000,B 0.000,C 90.000,E1 47.148} C_DIS
LIN {X -0.036,Y -253.836,Z 724.250,A 0.000,B 0.000,C 90.000,E1 45.000} C_DIS
LIN {X -0.112,Y -248.004,Z 724.238,A 0.000,B 0.000,C 90.000,E1 42.852} C_DIS
LIN {X 0.065,Y -242.062,Z 724.226,A 0.000,B 0.000,C 90.000,E1 40.620} C_DIS
LIN {X -0.101,Y -232.302,Z 724.205,A 0.000,B 0.000,C 90.000,E1 36.950} C_DIS
LIN {X -0.094,Y -223.298,Z 724.184,A 0.000,B 0.000,C 90.000,E1 33.166} C_DIS
LIN {X -0.057,Y -216.710,Z 724.167,A 0.000,B 0.000,C 90.000,E1 30.079} C_DIS
LIN {X -0.023,Y -210.859,Z 724.150,A 0.000,B 0.000,C 90.000,E1 26.950} C_DIS
LIN {X -0.049,Y -204.619,Z 724.128,A 0.000,B 0.000,C 90.000,E1 23.003} C_DIS
LIN {X -0.083,Y -200.513,Z 724.110,A 0.000,B 0.000,C 90.000,E1 19.812} C_DIS
LIN {X 0.050,Y -196.355,Z 724.087,A 0.000,B 0.000,C 90.000,E1 15.733} C_DIS
LIN {X 0.049,Y -192.793,Z 724.060,A 0.000,B 0.000,C 90.000,E1 10.838} C_DIS
LIN {X -0.092,Y -190.412,Z 724.024,A 0.000,B 0.000,C 90.000,E1 4.302} C_DIS
LIN {X -0.081,Y -191.820,Z 723.970,A 0.000,B 0.000,C 90.000,E1 354.609} C_DIS
LIN {X 0.080,Y -194.686,Z 723.943,A 0.000,B 0.000,C 90.000,E1 349.634} C_DIS
LIN {X 0.013,Y -198.214,Z 723.920,A 0.000,B 0.000,C 90.000,E1 345.574} C_DIS
LIN {X 0.012,Y -202.741,Z 723.897,A 0.000,B 0.000,C 90.000,E1 341.529} C_DIS
LIN {X -0.038,Y -208.140,Z 723.875,A 0.000,B 0.000,C 90.000,E1 337.539} C_DIS
LIN {X 0.034,Y -214.427,Z 723.853,A 0.000,B 0.000,C 90.000,E1 333.563} C_DIS
LIN {X 0.020,Y -221.298,Z 723.831,A 0.000,B 0.000,C 90.000,E1 329.665} C_DIS
LIN {X 0.040,Y -227.256,Z 723.814,A 0.000,B 0.000,C 90.000,E1 326.580} C_DIS
LIN {X 0.124,Y -235.244,Z 723.793,A 0.000,B 0.000,C 90.000,E1 322.763} C_DIS
LIN {X 0.013,Y -243.959,Z 723.773,A 0.000,B 0.000,C 90.000,E1 319.057} C_DIS
LIN {X -0.055,Y -253.604,Z 723.752,A 0.000,B 0.000,C 90.000,E1 315.405} C_DIS
LIN {X -0.158,Y -264.398,Z 723.732,A 0.000,B 0.000,C 90.000,E1 311.838} C_DIS
LIN {X -0.051,Y -276.267,Z 723.713,A 0.000,B 0.000,C 90.000,E1 308.302} C_DIS
LIN {X -0.028,Y -289.516,Z 723.694,A 0.000,B 0.000,C 90.000,E1 304.865} C_DIS
LIN {X 0.001,Y -304.304,Z 723.675,A 0.000,B 0.000,C 90.000,E1 301.514} C_DIS
LIN {X 0.088,Y -319.091,Z 723.659,A 0.000,B 0.000,C 90.000,E1 298.565} C_DIS
LIN {X -0.001,Y -337.168,Z 723.641,A 0.000,B 0.000,C 90.000,E1 295.412} C_DIS
LIN {X 0.006,Y -354.749,Z 723.626,A 0.000,B 0.000,C 90.000,E1 292.642} C_DIS
LIN {X 0.201,Y -375.564,Z 723.609,A 0.000,B 0.000,C 90.000,E1 289.631} C_DIS
LIN {X 0.175,Y -396.354,Z 723.595,A 0.000,B 0.000,C 90.000,E1 287.040} C_DIS
LIN {X 0.066,Y -410.480,Z 723.585,A 0.000,B 0.000,C 90.000,E1 285.371} C_DIS
LIN {X -0.044,Y -422.006,Z 723.578,A 0.000,B 0.000,C 90.000,E1 284.008} C_DIS
LIN {X 0.021,Y -433.395,Z 723.570,A 0.000,B 0.000,C 90.000,E1 282.647} C_DIS
LIN {X -0.061,Y -442.129,Z 723.564,A 0.000,B 0.000,C 90.000,E1 281.591} C_DIS
LIN {X 0.113,Y -452.542,Z 723.557,A 0.000,B 0.000,C 90.000,E1 280.254} C_DIS
LIN {X 0.045,Y -466.632,Z 723.547,A 0.000,B 0.000,C 90.000,E1 278.454} C_DIS
LIN {X -0.195,Y -474.192,Z 723.541,A 0.000,B 0.000,C 90.000,E1 277.466} C_DIS
LIN {X 0.193,Y -479.110,Z 723.537,A 0.000,B 0.000,C 90.000,E1 276.663} C_DIS
LIN {X 0.213,Y -483.255,Z 723.533,A 0.000,B 0.000,C 90.000,E1 275.910} C_DIS
LIN {X 0.215,Y -486.451,Z 723.529,A 0.000,B 0.000,C 90.000,E1 275.163} C_DIS
LIN {X -0.082,Y -488.059,Z 723.526,A 0.000,B 0.000,C 90.000,E1 274.702} C_DIS
LIN {X 0.079,Y -489.286,Z 723.523,A 0.000,B 0.000,C 90.000,E1 274.188} C_DIS
LIN {X -0.201,Y -490.045,Z 723.521,A 0.000,B 0.000,C 90.000,E1 273.726} C_DIS
LIN {X -0.016,Y -490.442,Z 723.518,A 0.000,B 0.000,C 90.000,E1 273.212} C_DIS
LIN {X 0.201,Y -490.463,Z 723.515,A 0.000,B 0.000,C 90.000,E1 272.694} C_DIS
LIN {X -0.094,Y -490.157,Z 723.512,A 0.000,B 0.000,C 90.000,E1 272.236} C_DIS
LIN {X 0.118,Y -489.497,Z 723.510,A 0.000,B 0.000,C 90.000,E1 271.718} C_DIS
LIN {X -0.176,Y -488.497,Z 723.507,A 0.000,B 0.000,C 90.000,E1 271.260} C_DIS
LIN {X 0.015,Y -487.067,Z 723.504,A 0.000,B 0.000,C 90.000,E1 270.745} C_DIS
LIN {X 0.199,Y -485.133,Z 723.501,A 0.000,B 0.000,C 90.000,E1 270.229} C_DIS
LIN {X -0.107,Y -482.665,Z 723.499,A 0.000,B 0.000,C 90.000,E1 269.771} C_DIS
LIN {X 0.051,Y -479.492,Z 723.496,A 0.000,B 0.000,C 90.000,E1 269.255} C_DIS
LIN {X 0.190,Y -475.443,Z 723.493,A 0.000,B 0.000,C 90.000,E1 268.740} C_DIS
LIN {X 0.012,Y -473.072,Z 723.492,A 0.000,B 0.000,C 90.000,E1 268.511} C_DIS
LIN {X -0.210,Y -467.593,Z 723.489,A 0.000,B 0.000,C 90.000,E1 268.051} C_DIS
LIN {X -0.062,Y -461.399,Z 723.487,A 0.000,B 0.000,C 90.000,E1 267.593} C_DIS
LIN {X 0.159,Y -454.638,Z 723.484,A 0.000,B 0.000,C 90.000,E1 267.192} C_DIS
LIN {X 0.027,Y -447.397,Z 723.483,A 0.000,B 0.000,C 90.000,E1 266.906} C_DIS
LIN {X -0.016,Y -439.795,Z 723.482,A 0.000,B 0.000,C 90.000,E1 266.674} C_DIS
LIN {X -0.031,Y -431.380,Z 723.481,A 0.000,B 0.000,C 90.000,E1 266.502} C_DIS
LIN {X -0.121,Y -426.218,Z 723.480,A 0.000,B 0.000,C 90.000,E1 266.445} C_DIS
LIN {X -0.081,Y -418.885,Z 723.480,A 0.000,B 0.000,C 90.000,E1 266.388} C_DIS
LIN {X -0.053,Y -180.940,Z 723.480,A 0.000,B 0.000,C 90.000,E1 266.388} C_DIS
LIN {X -0.047,Y -180.747,Z 723.470,A 0.000,B 0.000,C 90.000,E1 264.666} C_DIS
LIN {X 0.022,Y -178.838,Z 723.442,A 0.000,B 0.000,C 90.000,E1 259.577} C_DIS
LIN {X -0.082,Y -175.882,Z 723.414,A 0.000,B 0.000,C 90.000,E1 254.519} C_DIS
LIN {X 0.024,Y -174.547,Z 723.404,A 0.000,B 0.000,C 90.000,E1 252.779} C_DIS
LIN {X -0.043,Y -171.531,Z 723.381,A 0.000,B 0.000,C 90.000,E1 248.518} C_DIS
LIN {X -0.049,Y -167.757,Z 723.357,A 0.000,B 0.000,C 90.000,E1 244.204} C_DIS
LIN {X 0.040,Y -166.461,Z 723.347,A 0.000,B 0.000,C 90.000,E1 242.436} C_DIS
LIN {X 0.030,Y -163.176,Z 723.328,A 0.000,B 0.000,C 90.000,E1 238.948} C_DIS
LIN {X 0.079,Y -161.136,Z 723.313,A 0.000,B 0.000,C 90.000,E1 236.294} C_DIS
LIN {X -0.019,Y -157.157,Z 723.288,A 0.000,B 0.000,C 90.000,E1 231.904} C_DIS
LIN {X 0.004,Y -155.889,Z 723.278,A 0.000,B 0.000,C 90.000,E1 230.114} C_DIS
LIN {X -0.038,Y -152.138,Z 723.254,A 0.000,B 0.000,C 90.000,E1 225.648} C_DIS
LIN {X -0.017,Y -150.388,Z 723.238,A 0.000,B 0.000,C 90.000,E1 222.933} C_DIS
LIN {X 0.006,Y -147.120,Z 723.213,A 0.000,B 0.000,C 90.000,E1 218.382} C_DIS
LIN {X -0.002,Y -145.685,Z 723.198,A 0.000,B 0.000,C 90.000,E1 215.644} C_DIS
LIN {X -0.004,Y -143.067,Z 723.172,A 0.000,B 0.000,C 90.000,E1 211.052} C_DIS
LIN {X -0.073,Y -141.688,Z 723.152,A 0.000,B 0.000,C 90.000,E1 207.385} C_DIS
LIN {X -0.018,Y -139.460,Z 723.116,A 0.000,B 0.000,C 90.000,E1 200.865} C_DIS
LIN {X 0.082,Y -139.194,Z 723.106,A 0.000,B 0.000,C 90.000,E1 198.960} C_DIS
LIN {X -0.032,Y -138.325,Z 723.054,A 0.000,B 0.000,C 90.000,E1 189.670} C_DIS
LIN {X -0.027,Y -139.452,Z 723.007,A 0.000,B 0.000,C 90.000,E1 181.260} C_DIS
LIN {X 0.053,Y -140.998,Z 722.976,A 0.000,B 0.000,C 90.000,E1 175.641} C_DIS
LIN {X 0.003,Y -142.753,Z 722.955,A 0.000,B 0.000,C 90.000,E1 171.951} C_DIS
LIN {X -0.041,Y -145.153,Z 722.930,A 0.000,B 0.000,C 90.000,E1 167.353} C_DIS
LIN {X -0.048,Y -147.775,Z 722.909,A 0.000,B 0.000,C 90.000,E1 163.685} C_DIS
LIN {X 0.031,Y -150.452,Z 722.889,A 0.000,B 0.000,C 90.000,E1 160.007} C_DIS
LIN {X -0.034,Y -153.901,Z 722.869,A 0.000,B 0.000,C 90.000,E1 156.410} C_DIS
LIN {X 0.031,Y -157.312,Z 722.849,A 0.000,B 0.000,C 90.000,E1 152.794} C_DIS
LIN {X -0.022,Y -161.498,Z 722.829,A 0.000,B 0.000,C 90.000,E1 149.253} C_DIS
LIN {X -0.007,Y -165.698,Z 722.810,A 0.000,B 0.000,C 90.000,E1 145.722} C_DIS
LIN {X -0.016,Y -170.641,Z 722.790,A 0.000,B 0.000,C 90.000,E1 142.236} C_DIS
LIN {X 0.032,Y -175.517,Z 722.771,A 0.000,B 0.000,C 90.000,E1 138.771} C_DIS
LIN {X -0.102,Y -181.137,Z 722.752,A 0.000,B 0.000,C 90.000,E1 135.405} C_DIS
LIN {X 0.025,Y -186.588,Z 722.733,A 0.000,B 0.000,C 90.000,E1 132.000} C_DIS
LIN {X -0.009,Y -191.584,Z 722.718,A 0.000,B 0.000,C 90.000,E1 129.277} C_DIS
LIN {X -0.063,Y -290.214,Z 722.718,A 0.000,B 0.000,C 90.000,E1 129.277} C_DIS
LIN {X -0.026,Y -291.958,Z 722.718,A 0.000,B 0.000,C 90.000,E1 129.241} C_DIS
LIN {X 0.029,Y -297.243,Z 722.716,A 0.000,B 0.000,C 90.000,E1 128.955} C_DIS
LIN {X 0.085,Y -300.031,Z 722.715,A 0.000,B 0.000,C 90.000,E1 128.669} C_DIS
LIN {X 0.144,Y -303.733,Z 722.712,A 0.000,B 0.000,C 90.000,E1 128.096} C_DIS
LIN {X -0.092,Y -305.255,Z 722.710,A 0.000,B 0.000,C 90.000,E1 127.810} C_DIS
LIN {X 0.101,Y -306.451,Z 722.708,A 0.000,B 0.000,C 90.000,E1 127.443} C_DIS
LIN {X 0.086,Y -317.169,Z 722.688,A 0.000,B 0.000,C 90.000,E1 123.865} C_DIS
LIN {X 0.015,Y -327.263,Z 722.672,A 0.000,B 0.000,C 90.000,E1 121.003} C_DIS
LIN {X 0.015,Y -338.683,Z 722.657,A 0.000,B 0.000,C 90.000,E1 118.180} C_DIS
LIN {X 0.023,Y -351.539,Z 722.641,A 0.000,B 0.000,C 90.000,E1 115.412} C_DIS
LIN {X -0.124,Y -364.259,Z 722.628,A 0.000,B 0.000,C 90.000,E1 113.025} C_DIS
LIN {X -0.106,Y -378.293,Z 722.615,A 0.000,B 0.000,C 90.000,E1 110.663} C_DIS
LIN {X -0.142,Y -393.740,Z 722.602,A 0.000,B 0.000,C 90.000,E1 108.362} C_DIS
LIN {X 0.093,Y -410.713,Z 722.589,A 0.000,B 0.000,C 90.000,E1 106.079} C_DIS
LIN {X 0.133,Y -429.337,Z 722.577,A 0.000,B 0.000,C 90.000,E1 103.883} C_DIS
LIN {X -0.089,Y -449.292,Z 722.566,A 0.000,B 0.000,C 90.000,E1 101.827} C_DIS
LIN {X -0.056,Y -467.210,Z 722.556,A 0.000,B 0.000,C 90.000,E1 100.141} C_DIS
LIN {X -0.022,Y -469.528,Z 722.555,A 0.000,B 0.000,C 90.000,E1 99.905} C_DIS
LIN {X -0.120,Y -471.378,Z 722.554,A 0.000,B 0.000,C 90.000,E1 99.670} C_DIS
LIN {X 0.247,Y -472.776,Z 722.552,A 0.000,B 0.000,C 90.000,E1 99.378} C_DIS
LIN {X -0.115,Y -474.608,Z 722.549,A 0.000,B 0.000,C 90.000,E1 98.916} C_DIS
LIN {X 0.001,Y -475.345,Z 722.547,A 0.000,B 0.000,C 90.000,E1 98.398} C_DIS
LIN {X 0.195,Y -475.111,Z 722.544,A 0.000,B 0.000,C 90.000,E1 97.871} C_DIS
LIN {X -0.143,Y -473.876,Z 722.541,A 0.000,B 0.000,C 90.000,E1 97.409} C_DIS
LIN {X 0.127,Y -472.825,Z 722.540,A 0.000,B 0.000,C 90.000,E1 97.125} C_DIS
LIN {X -0.012,Y -471.416,Z 722.538,A 0.000,B 0.000,C 90.000,E1 96.891} C_DIS
LIN {X 0.105,Y -453.482,Z 722.523,A 0.000,B 0.000,C 90.000,E1 94.073} C_DIS
LIN {X 0.187,Y -440.125,Z 722.510,A 0.000,B 0.000,C 90.000,E1 91.718} C_DIS
LIN {X -0.128,Y -431.148,Z 722.501,A 0.000,B 0.000,C 90.000,E1 90.172} C_DIS
SetRPM(0)
End
